   instHMIStationDriver.instsHSSPartSelect[2].lib.raw[9,5] := WSTRING#'16.18.011.321.010A';
   instHMIStationDriver.instsHSSPartSelect[2].lib.raw[9,6] := WSTRING#'16.18.008.301.030A';
   instHMIStationDriver.instsHSSPartSelect[2].lib.raw[9,7] := WSTRING#'16.18.011.321.020B';
   instHMIStationDriver.instsHSSPartSelect[2].lib.raw[10,0] := WSTRING#'';
   instHMIStationDriver.instsHSSPartSelect[2].lib.raw[10,1] := WSTRING#'C/O MATERIALS';
   instHMIStationDriver.instsHSSPartSelect[2].lib.raw[10,2] := WSTRING#'16.18.007.301.010A';
   instHMIStationDriver.instsHSSPartSelect[2].lib.raw[10,3] := WSTRING#'16.18.011.321.020B';
   instHMIStationDriver.instsHSSPartSelect[2].lib.raw[10,4] := WSTRING#'';
   instHMIStationDriver.instsHSSPartSelect[2].lib.raw[10,5] := WSTRING#'16.18.008.301.020A';
   instHMIStationDriver.instsHSSPartSelect[2].lib.raw[10,6] := WSTRING#'16.18.008.301.030A';
   instHMIStationDriver.instsHSSPartSelect[2].lib.raw[10,7] := WSTRING#'16.18.011.301.020B';
   instHMIStationDriver.instsHSSPartSelect[2].lib.raw[11,0] := WSTRING#'';
   instHMIStationDriver.instsHSSPartSelect[2].lib.raw[11,1] := WSTRING#'C/O MATERIALS';
   instHMIStationDriver.instsHSSPartSelect[2].lib.raw[11,2] := WSTRING#'16.18.008.311.010A';
   instHMIStationDriver.instsHSSPartSelect[2].lib.raw[11,3] := WSTRING#'';
   instHMIStationDriver.instsHSSPartSelect[2].lib.raw[11,4] := WSTRING#'';
   instHMIStationDriver.instsHSSPartSelect[2].lib.raw[11,5] := WSTRING#'';
   instHMIStationDriver.instsHSSPartSelect[2].lib.raw[11,6] := WSTRING#'16.18.008.301.030A';
   instHMIStationDriver.instsHSSPartSelect[2].lib.raw[11,7] := WSTRING#'16.18.008.311.020B';
   instHMIStationDriver.instsHSSPartSelect[2].lib.raw[12,0] := WSTRING#'';
   instHMIStationDriver.instsHSSPartSelect[2].lib.raw[12,1] := WSTRING#'C/O MATERIALS';
   instHMIStationDriver.instsHSSPartSelect[2].lib.raw[12,2] := WSTRING#'16.18.009.301.010A';
   instHMIStationDriver.instsHSSPartSelect[2].lib.raw[12,3] := WSTRING#'16.18.009.301.040B';
   instHMIStationDriver.instsHSSPartSelect[2].lib.raw[12,4] := WSTRING#'';
   instHMIStationDriver.instsHSSPartSelect[2].lib.raw[12,5] := WSTRING#'16.18.009.301.030A';
   instHMIStationDriver.instsHSSPartSelect[2].lib.raw[12,6] := WSTRING#'16.18.009.301.050A';
   instHMIStationDriver.instsHSSPartSelect[2].lib.raw[12,7] := WSTRING#'16.18.009.301.020B';
   instHMIStationDriver.instsHSSPartSelect[2].lib.raw[13,0] := WSTRING#'';
   instHMIStationDriver.instsHSSPartSelect[2].lib.raw[13,1] := WSTRING#'C/O MATERIALS';
   instHMIStationDriver.instsHSSPartSelect[2].lib.raw[13,2] := WSTRING#'16.18.009.311.010A';
   instHMIStationDriver.instsHSSPartSelect[2].lib.raw[13,3] := WSTRING#'';
   instHMIStationDriver.instsHSSPartSelect[2].lib.raw[13,4] := WSTRING#'';
   instHMIStationDriver.instsHSSPartSelect[2].lib.raw[13,5] := WSTRING#'16.18.009.301.030A';
   instHMIStationDriver.instsHSSPartSelect[2].lib.raw[13,6] := WSTRING#'16.18.009.301.050A';
   instHMIStationDriver.instsHSSPartSelect[2].lib.raw[13,7] := WSTRING#'16.18.009.301.040B';
   instHMIStationDriver.instsHSSPartSelect[2].lib.raw[14,0] := WSTRING#'';
   instHMIStationDriver.instsHSSPartSelect[2].lib.raw[14,1] := WSTRING#'C/O MATERIALS';
   instHMIStationDriver.instsHSSPartSelect[2].lib.raw[14,2] := WSTRING#'16.18.009.321.010A';
   instHMIStationDriver.instsHSSPartSelect[2].lib.raw[14,3] := WSTRING#'16.18.009.301.020B';
   instHMIStationDriver.instsHSSPartSelect[2].lib.raw[14,4] := WSTRING#'';
   instHMIStationDriver.instsHSSPartSelect[2].lib.raw[14,5] := WSTRING#'16.18.009.321.030A';
   instHMIStationDriver.instsHSSPartSelect[2].lib.raw[14,6] := WSTRING#'16.18.009.301.050A';
   instHMIStationDriver.instsHSSPartSelect[2].lib.raw[14,7] := WSTRING#'16.18.009.321.020B';
   instHMIStationDriver.instsHSSPartSelect[2].lib.raw[15,0] := WSTRING#'';
   instHMIStationDriver.instsHSSPartSelect[2].lib.raw[15,1] := WSTRING#'C/O MATERIALS';
   instHMIStationDriver.instsHSSPartSelect[2].lib.raw[15,2] := WSTRING#'16.18.009.321.010A';
   instHMIStationDriver.instsHSSPartSelect[2].lib.raw[15,3] := WSTRING#'16.18.009.321.020B';
   instHMIStationDriver.instsHSSPartSelect[2].lib.raw[15,4] := WSTRING#'';
   instHMIStationDriver.instsHSSPartSelect[2].lib.raw[15,5] := WSTRING#'16.18.009.321.030A';
   instHMIStationDriver.instsHSSPartSelect[2].lib.raw[15,6] := WSTRING#'16.18.009.331.050A';
   instHMIStationDriver.instsHSSPartSelect[2].lib.raw[15,7] := WSTRING#'16.18.009.301.020B';
   instHMIStationDriver.instsHSSPartSelect[2].lib.raw[16,0] := WSTRING#'';
   instHMIStationDriver.instsHSSPartSelect[2].lib.raw[16,1] := WSTRING#'C/O MATERIALS';
   instHMIStationDriver.instsHSSPartSelect[2].lib.raw[16,2] := WSTRING#'16.18.009.331.030A';
   instHMIStationDriver.instsHSSPartSelect[2].lib.raw[16,3] := WSTRING#'';
   instHMIStationDriver.instsHSSPartSelect[2].lib.raw[16,4] := WSTRING#'';
   instHMIStationDriver.instsHSSPartSelect[2].lib.raw[16,5] := WSTRING#'16.18.009.371.010A';
   instHMIStationDriver.instsHSSPartSelect[2].lib.raw[16,6] := WSTRING#'16.18.009.301.050A';
   instHMIStationDriver.instsHSSPartSelect[2].lib.raw[16,7] := WSTRING#'16.18.009.301.020B';
   instHMIStationDriver.instsHSSPartSelect[2].lib.raw[17,0] := WSTRING#'';
   instHMIStationDriver.instsHSSPartSelect[2].lib.raw[17,1] := WSTRING#'C/O MATERIALS';
   instHMIStationDriver.instsHSSPartSelect[2].lib.raw[17,2] := WSTRING#'16.18.011.301.030A';
   instHMIStationDriver.instsHSSPartSelect[2].lib.raw[17,3] := WSTRING#'16.18.011.301.040B';
   instHMIStationDriver.instsHSSPartSelect[2].lib.raw[17,4] := WSTRING#'';
   instHMIStationDriver.instsHSSPartSelect[2].lib.raw[17,5] := WSTRING#'16.18.011.301.010A';
   instHMIStationDriver.instsHSSPartSelect[2].lib.raw[17,6] := WSTRING#'16.18.008.301.030A';
   instHMIStationDriver.instsHSSPartSelect[2].lib.raw[17,7] := WSTRING#'16.18.011.301.020B';
   instHMIStationDriver.instsHSSPartSelect[2].lib.raw[18,0] := WSTRING#'';
   instHMIStationDriver.instsHSSPartSelect[2].lib.raw[18,1] := WSTRING#'C/O MATERIALS';
   instHMIStationDriver.instsHSSPartSelect[2].lib.raw[18,2] := WSTRING#'16.18.007.301.010A';
   instHMIStationDriver.instsHSSPartSelect[2].lib.raw[18,3] := WSTRING#'';
   instHMIStationDriver.instsHSSPartSelect[2].lib.raw[18,4] := WSTRING#'';
   instHMIStationDriver.instsHSSPartSelect[2].lib.raw[18,5] := WSTRING#'16.18.011.321.010A';
   instHMIStationDriver.instsHSSPartSelect[2].lib.raw[18,6] := WSTRING#'16.18.011.311.020A';
   instHMIStationDriver.instsHSSPartSelect[2].lib.raw[18,7] := WSTRING#'16.18.011.321.020B';
   instHMIStationDriver.instsHSSPartSelect[2].lib.raw[19,0] := WSTRING#'';
   instHMIStationDriver.instsHSSPartSelect[2].lib.raw[19,1] := WSTRING#'C/O MATERIALS';
   instHMIStationDriver.instsHSSPartSelect[2].lib.raw[19,2] := WSTRING#'16.18.011.321.010A';
   instHMIStationDriver.instsHSSPartSelect[2].lib.raw[19,3] := WSTRING#'16.18.011.301.020B';
   instHMIStationDriver.instsHSSPartSelect[2].lib.raw[19,4] := WSTRING#'';
   instHMIStationDriver.instsHSSPartSelect[2].lib.raw[19,5] := WSTRING#'16.18.011.301.010A';
   instHMIStationDriver.instsHSSPartSelect[2].lib.raw[19,6] := WSTRING#'16.18.011.321.030A';
   instHMIStationDriver.instsHSSPartSelect[2].lib.raw[19,7] := WSTRING#'16.18.011.321.020B';
   instHMIStationDriver.instsHSSPartSelect[2].lib.raw[20,0] := WSTRING#'';
   instHMIStationDriver.instsHSSPartSelect[2].lib.raw[20,1] := WSTRING#'C/O MATERIALS';
   instHMIStationDriver.instsHSSPartSelect[2].lib.raw[20,2] := WSTRING#'16.18.011.331.010A';
   instHMIStationDriver.instsHSSPartSelect[2].lib.raw[20,3] := WSTRING#'';
   instHMIStationDriver.instsHSSPartSelect[2].lib.raw[20,4] := WSTRING#'';
   instHMIStationDriver.instsHSSPartSelect[2].lib.raw[20,5] := WSTRING#'';
   instHMIStationDriver.instsHSSPartSelect[2].lib.raw[20,6] := WSTRING#'16.18.011.311.020A';
   instHMIStationDriver.instsHSSPartSelect[2].lib.raw[20,7] := WSTRING#'16.18.011.331.020D';
   instHMIStationDriver.instsHSSPartSelect[2].lib.raw[21,0] := WSTRING#'';
   instHMIStationDriver.instsHSSPartSelect[2].lib.raw[21,1] := WSTRING#'C/O MATERIALS';
   instHMIStationDriver.instsHSSPartSelect[2].lib.raw[21,2] := WSTRING#'16.18.012.401.010A';
   instHMIStationDriver.instsHSSPartSelect[2].lib.raw[21,3] := WSTRING#'';
   instHMIStationDriver.instsHSSPartSelect[2].lib.raw[21,4] := WSTRING#'';
   instHMIStationDriver.instsHSSPartSelect[2].lib.raw[21,5] := WSTRING#'';
   instHMIStationDriver.instsHSSPartSelect[2].lib.raw[21,6] := WSTRING#'16.18.014.411.030A';
   instHMIStationDriver.instsHSSPartSelect[2].lib.raw[21,7] := WSTRING#'16.18.012.401.020A';
   instHMIStationDriver.instsHSSPartSelect[2].lib.raw[22,0] := WSTRING#'';
   instHMIStationDriver.instsHSSPartSelect[2].lib.raw[22,1] := WSTRING#'C/O MATERIALS';
   instHMIStationDriver.instsHSSPartSelect[2].lib.raw[22,2] := WSTRING#'16.18.012.411.010A';
   instHMIStationDriver.instsHSSPartSelect[2].lib.raw[22,3] := WSTRING#'';
   instHMIStationDriver.instsHSSPartSelect[2].lib.raw[22,4] := WSTRING#'';
   instHMIStationDriver.instsHSSPartSelect[2].lib.raw[22,5] := WSTRING#'';
   instHMIStationDriver.instsHSSPartSelect[2].lib.raw[22,6] := WSTRING#'16.18.014.411.030A';
   instHMIStationDriver.instsHSSPartSelect[2].lib.raw[22,7] := WSTRING#'16.18.012.411.020B';
   instHMIStationDriver.instsHSSPartSelect[2].lib.raw[23,0] := WSTRING#'';
   instHMIStationDriver.instsHSSPartSelect[2].lib.raw[23,1] := WSTRING#'C/O MATERIALS';
   instHMIStationDriver.instsHSSPartSelect[2].lib.raw[23,2] := WSTRING#'16.18.014.411.010A';
   instHMIStationDriver.instsHSSPartSelect[2].lib.raw[23,3] := WSTRING#'';
   instHMIStationDriver.instsHSSPartSelect[2].lib.raw[23,4] := WSTRING#'';
   instHMIStationDriver.instsHSSPartSelect[2].lib.raw[23,5] := WSTRING#'';
   instHMIStationDriver.instsHSSPartSelect[2].lib.raw[23,6] := WSTRING#'16.18.014.411.030A';
   instHMIStationDriver.instsHSSPartSelect[2].lib.raw[23,7] := WSTRING#'16.18.012.401.020A';
   instHMIStationDriver.instsHSSPartSelect[2].lib.raw[24,0] := WSTRING#'';
   instHMIStationDriver.instsHSSPartSelect[2].lib.raw[24,1] := WSTRING#'C/O MATERIALS';
   instHMIStationDriver.instsHSSPartSelect[2].lib.raw[24,2] := WSTRING#'16.18.012.431.010A';
   instHMIStationDriver.instsHSSPartSelect[2].lib.raw[24,3] := WSTRING#'';
   instHMIStationDriver.instsHSSPartSelect[2].lib.raw[24,4] := WSTRING#'';
   instHMIStationDriver.instsHSSPartSelect[2].lib.raw[24,5] := WSTRING#'';
   instHMIStationDriver.instsHSSPartSelect[2].lib.raw[24,6] := WSTRING#'16.18.014.411.030A';
   instHMIStationDriver.instsHSSPartSelect[2].lib.raw[24,7] := WSTRING#'16.18.012.411.020B';
   instHMIStationDriver.instsHSSPartSelect[2].lib.raw[25,0] := WSTRING#'';
   instHMIStationDriver.instsHSSPartSelect[2].lib.raw[25,1] := WSTRING#'C/O MATERIALS';
   instHMIStationDriver.instsHSSPartSelect[2].lib.raw[25,2] := WSTRING#'16.18.012.441.010A';
   instHMIStationDriver.instsHSSPartSelect[2].lib.raw[25,3] := WSTRING#'';
   instHMIStationDriver.instsHSSPartSelect[2].lib.raw[25,4] := WSTRING#'';
   instHMIStationDriver.instsHSSPartSelect[2].lib.raw[25,5] := WSTRING#'';
   instHMIStationDriver.instsHSSPartSelect[2].lib.raw[25,6] := WSTRING#'16.18.013.411.030A';
   instHMIStationDriver.instsHSSPartSelect[2].lib.raw[25,7] := WSTRING#'16.18.011.321.020B';
   instHMIStationDriver.instsHSSPartSelect[2].lib.raw[26,0] := WSTRING#'';
   instHMIStationDriver.instsHSSPartSelect[2].lib.raw[26,1] := WSTRING#'C/O MATERIALS';
   instHMIStationDriver.instsHSSPartSelect[2].lib.raw[26,2] := WSTRING#'16.18.013.411.010A';
   instHMIStationDriver.instsHSSPartSelect[2].lib.raw[26,3] := WSTRING#'';
   instHMIStationDriver.instsHSSPartSelect[2].lib.raw[26,4] := WSTRING#'';
   instHMIStationDriver.instsHSSPartSelect[2].lib.raw[26,5] := WSTRING#'';
   instHMIStationDriver.instsHSSPartSelect[2].lib.raw[26,6] := WSTRING#'16.18.013.411.030A';
   instHMIStationDriver.instsHSSPartSelect[2].lib.raw[26,7] := WSTRING#'16.18.013.411.020B';
   instHMIStationDriver.instsHSSPartSelect[2].lib.raw[27,0] := WSTRING#'';
   instHMIStationDriver.instsHSSPartSelect[2].lib.raw[27,1] := WSTRING#'C/O MATERIALS';
   instHMIStationDriver.instsHSSPartSelect[2].lib.raw[27,2] := WSTRING#'16.18.013.421.010A';
   instHMIStationDriver.instsHSSPartSelect[2].lib.raw[27,3] := WSTRING#'';
   instHMIStationDriver.instsHSSPartSelect[2].lib.raw[27,4] := WSTRING#'';
   instHMIStationDriver.instsHSSPartSelect[2].lib.raw[27,5] := WSTRING#'';
   instHMIStationDriver.instsHSSPartSelect[2].lib.raw[27,6] := WSTRING#'16.18.013.411.030A';
   instHMIStationDriver.instsHSSPartSelect[2].lib.raw[27,7] := WSTRING#'16.18.011.301.040B';
   instHMIStationDriver.instsHSSPartSelect[2].lib.raw[28,0] := WSTRING#'';
   instHMIStationDriver.instsHSSPartSelect[2].lib.raw[28,1] := WSTRING#'C/O MATERIALS';
   instHMIStationDriver.instsHSSPartSelect[2].lib.raw[28,2] := WSTRING#'16.18.015.421.010A';
   instHMIStationDriver.instsHSSPartSelect[2].lib.raw[28,3] := WSTRING#'';
   instHMIStationDriver.instsHSSPartSelect[2].lib.raw[28,4] := WSTRING#'';
   instHMIStationDriver.instsHSSPartSelect[2].lib.raw[28,5] := WSTRING#'';
   instHMIStationDriver.instsHSSPartSelect[2].lib.raw[28,6] := WSTRING#'16.18.015.401.010A';
   instHMIStationDriver.instsHSSPartSelect[2].lib.raw[28,7] := WSTRING#'16.18.015.421.020B';
   instHMIStationDriver.instsHSSPartSelect[2].lib.raw[29,0] := WSTRING#'';
   instHMIStationDriver.instsHSSPartSelect[2].lib.raw[29,1] := WSTRING#'C/O MATERIALS';
   instHMIStationDriver.instsHSSPartSelect[2].lib.raw[29,2] := WSTRING#'16.18.015.411.010A';
   instHMIStationDriver.instsHSSPartSelect[2].lib.raw[29,3] := WSTRING#'';
   instHMIStationDriver.instsHSSPartSelect[2].lib.raw[29,4] := WSTRING#'';
   instHMIStationDriver.instsHSSPartSelect[2].lib.raw[29,5] := WSTRING#'';
   instHMIStationDriver.instsHSSPartSelect[2].lib.raw[29,6] := WSTRING#'16.18.015.411.030A';
   instHMIStationDriver.instsHSSPartSelect[2].lib.raw[29,7] := WSTRING#'16.18.015.411.020B';
   instHMIStationDriver.instsHSSPartSelect[2].lib.raw[30,0] := WSTRING#'';
   instHMIStationDriver.instsHSSPartSelect[2].lib.raw[30,1] := WSTRING#'C/O MATERIALS';
   instHMIStationDriver.instsHSSPartSelect[2].lib.raw[30,2] := WSTRING#'16.18.018.401.010A';
   instHMIStationDriver.instsHSSPartSelect[2].lib.raw[30,3] := WSTRING#'';
   instHMIStationDriver.instsHSSPartSelect[2].lib.raw[30,4] := WSTRING#'';
   instHMIStationDriver.instsHSSPartSelect[2].lib.raw[30,5] := WSTRING#'';
   instHMIStationDriver.instsHSSPartSelect[2].lib.raw[30,6] := WSTRING#'16.18.015.401.010A';
   instHMIStationDriver.instsHSSPartSelect[2].lib.raw[30,7] := WSTRING#'16.18.018.401.020B';
   instHMIStationDriver.instsHSSPartSelect[2].lib.raw[31,0] := WSTRING#'';
   instHMIStationDriver.instsHSSPartSelect[2].lib.raw[31,1] := WSTRING#'C/O MATERIALS';
   instHMIStationDriver.instsHSSPartSelect[2].lib.raw[31,2] := WSTRING#'16.18.018.421.010B';
   instHMIStationDriver.instsHSSPartSelect[2].lib.raw[31,3] := WSTRING#'';
   instHMIStationDriver.instsHSSPartSelect[2].lib.raw[31,4] := WSTRING#'';
   instHMIStationDriver.instsHSSPartSelect[2].lib.raw[31,5] := WSTRING#'';
   instHMIStationDriver.instsHSSPartSelect[2].lib.raw[31,6] := WSTRING#'16.18.015.411.030A';
   instHMIStationDriver.instsHSSPartSelect[2].lib.raw[31,7] := WSTRING#'16.18.015.411.020B';
   instHMIStationDriver.instsHSSPartSelect[2].lib.raw[32,0] := WSTRING#'';
   instHMIStationDriver.instsHSSPartSelect[2].lib.raw[32,1] := WSTRING#'C/O MATERIALS';
   instHMIStationDriver.instsHSSPartSelect[2].lib.raw[32,2] := WSTRING#'16.18.018.401.010A';
   instHMIStationDriver.instsHSSPartSelect[2].lib.raw[32,3] := WSTRING#'';
   instHMIStationDriver.instsHSSPartSelect[2].lib.raw[32,4] := WSTRING#'';
   instHMIStationDriver.instsHSSPartSelect[2].lib.raw[32,5] := WSTRING#'';
   instHMIStationDriver.instsHSSPartSelect[2].lib.raw[32,6] := WSTRING#'16.18.015.411.030A';
   instHMIStationDriver.instsHSSPartSelect[2].lib.raw[32,7] := WSTRING#'16.18.018.401.020B';
   instHMIStationDriver.instsHSSPartSelect[2].lib.raw[33,0] := WSTRING#'';
   instHMIStationDriver.instsHSSPartSelect[2].lib.raw[33,1] := WSTRING#'C/O MATERIALS';
   instHMIStationDriver.instsHSSPartSelect[2].lib.raw[33,2] := WSTRING#'16.18.017.301.030A';
   instHMIStationDriver.instsHSSPartSelect[2].lib.raw[33,3] := WSTRING#'16.18.017.301.020A';
   instHMIStationDriver.instsHSSPartSelect[2].lib.raw[33,4] := WSTRING#'';
   instHMIStationDriver.instsHSSPartSelect[2].lib.raw[33,5] := WSTRING#'16.18.017.301.010A';
   instHMIStationDriver.instsHSSPartSelect[2].lib.raw[33,6] := WSTRING#'16.18.017.301.050A';
   instHMIStationDriver.instsHSSPartSelect[2].lib.raw[33,7] := WSTRING#'16.18.017.301.040A';
   instHMIStationDriver.instsHSSPartSelect[2].lib.raw[34,0] := WSTRING#'';
   instHMIStationDriver.instsHSSPartSelect[2].lib.raw[34,1] := WSTRING#'C/O MATERIALS';
   instHMIStationDriver.instsHSSPartSelect[2].lib.raw[34,2] := WSTRING#'16.18.017.301.030A';
   instHMIStationDriver.instsHSSPartSelect[2].lib.raw[34,3] := WSTRING#'';
   instHMIStationDriver.instsHSSPartSelect[2].lib.raw[34,4] := WSTRING#'';
   instHMIStationDriver.instsHSSPartSelect[2].lib.raw[34,5] := WSTRING#'16.18.017.311.010A';
   instHMIStationDriver.instsHSSPartSelect[2].lib.raw[34,6] := WSTRING#'16.18.017.301.050A';
   instHMIStationDriver.instsHSSPartSelect[2].lib.raw[34,7] := WSTRING#'16.18.017.301.040A';
   instHMIStationDriver.instsHSSPartSelect[2].lib.raw[35,0] := WSTRING#'';
   instHMIStationDriver.instsHSSPartSelect[2].lib.raw[35,1] := WSTRING#'C/O MATERIALS';
   instHMIStationDriver.instsHSSPartSelect[2].lib.raw[35,2] := WSTRING#'16.18.017.321.010A';
   instHMIStationDriver.instsHSSPartSelect[2].lib.raw[35,3] := WSTRING#'';
   instHMIStationDriver.instsHSSPartSelect[2].lib.raw[35,4] := WSTRING#'';
   instHMIStationDriver.instsHSSPartSelect[2].lib.raw[35,5] := WSTRING#'';
   instHMIStationDriver.instsHSSPartSelect[2].lib.raw[35,6] := WSTRING#'16.18.017.301.050A';
   instHMIStationDriver.instsHSSPartSelect[2].lib.raw[35,7] := WSTRING#'16.18.017.321.020A';
   instHMIStationDriver.instsHSSPartSelect[2].lib.raw[36,0] := WSTRING#'';
   instHMIStationDriver.instsHSSPartSelect[2].lib.raw[36,1] := WSTRING#'C/O MATERIALS';
   instHMIStationDriver.instsHSSPartSelect[2].lib.raw[36,2] := WSTRING#'16.18.018.401.010A';
   instHMIStationDriver.instsHSSPartSelect[2].lib.raw[36,3] := WSTRING#'';
   instHMIStationDriver.instsHSSPartSelect[2].lib.raw[36,4] := WSTRING#'';
   instHMIStationDriver.instsHSSPartSelect[2].lib.raw[36,5] := WSTRING#'';
   instHMIStationDriver.instsHSSPartSelect[2].lib.raw[36,6] := WSTRING#'16.18.018.401.030A';
   instHMIStationDriver.instsHSSPartSelect[2].lib.raw[36,7] := WSTRING#'16.18.018.401.020B';
   instHMIStationDriver.instsHSSPartSelect[2].lib.raw[37,0] := WSTRING#'';
   instHMIStationDriver.instsHSSPartSelect[2].lib.raw[37,1] := WSTRING#'C/O MATERIALS';
   instHMIStationDriver.instsHSSPartSelect[2].lib.raw[37,2] := WSTRING#'16.18.015.411.010A';
   instHMIStationDriver.instsHSSPartSelect[2].lib.raw[37,3] := WSTRING#'';
   instHMIStationDriver.instsHSSPartSelect[2].lib.raw[37,4] := WSTRING#'';
   instHMIStationDriver.instsHSSPartSelect[2].lib.raw[37,5] := WSTRING#'';
   instHMIStationDriver.instsHSSPartSelect[2].lib.raw[37,6] := WSTRING#'16.18.018.401.030A';
   instHMIStationDriver.instsHSSPartSelect[2].lib.raw[37,7] := WSTRING#'16.18.015.411.020B';
   instHMIStationDriver.instsHSSPartSelect[2].lib.raw[38,0] := WSTRING#'';
   instHMIStationDriver.instsHSSPartSelect[2].lib.raw[38,1] := WSTRING#'C/O MATERIALS';
   instHMIStationDriver.instsHSSPartSelect[2].lib.raw[38,2] := WSTRING#'16.18.018.411.010A';
   instHMIStationDriver.instsHSSPartSelect[2].lib.raw[38,3] := WSTRING#'';
   instHMIStationDriver.instsHSSPartSelect[2].lib.raw[38,4] := WSTRING#'';
   instHMIStationDriver.instsHSSPartSelect[2].lib.raw[38,5] := WSTRING#'';
   instHMIStationDriver.instsHSSPartSelect[2].lib.raw[38,6] := WSTRING#'16.18.018.401.030A';
   instHMIStationDriver.instsHSSPartSelect[2].lib.raw[38,7] := WSTRING#'16.18.018.401.020B';
   instHMIStationDriver.instsHSSPartSelect[2].lib.raw[39,0] := WSTRING#'';
   instHMIStationDriver.instsHSSPartSelect[2].lib.raw[39,1] := WSTRING#'C/O MATERIALS';
   instHMIStationDriver.instsHSSPartSelect[2].lib.raw[39,2] := WSTRING#'16.18.018.421.010B';
   instHMIStationDriver.instsHSSPartSelect[2].lib.raw[39,3] := WSTRING#'';
   instHMIStationDriver.instsHSSPartSelect[2].lib.raw[39,4] := WSTRING#'';
   instHMIStationDriver.instsHSSPartSelect[2].lib.raw[39,5] := WSTRING#'';
   instHMIStationDriver.instsHSSPartSelect[2].lib.raw[39,6] := WSTRING#'16.18.018.401.030A';
   instHMIStationDriver.instsHSSPartSelect[2].lib.raw[39,7] := WSTRING#'16.18.015.411.020B';
   instHMIStationDriver.instsHSSPartSelect[2].lib.raw[40,0] := WSTRING#'';
   instHMIStationDriver.instsHSSPartSelect[2].lib.raw[40,1] := WSTRING#'C/O MATERIALS';
   instHMIStationDriver.instsHSSPartSelect[2].lib.raw[40,2] := WSTRING#'16.18.008.301.010A';
   instHMIStationDriver.instsHSSPartSelect[2].lib.raw[40,3] := WSTRING#'16.18.011.321.020B';
   instHMIStationDriver.instsHSSPartSelect[2].lib.raw[40,4] := WSTRING#'';
   instHMIStationDriver.instsHSSPartSelect[2].lib.raw[40,5] := WSTRING#'16.18.011.321.010A';
   instHMIStationDriver.instsHSSPartSelect[2].lib.raw[40,6] := WSTRING#'16.18.011.311.020A';
   instHMIStationDriver.instsHSSPartSelect[2].lib.raw[40,7] := WSTRING#'16.18.012.401.020A';
   instHMIStationDriver.instsHSSPartSelect[2].lib.raw[41,0] := WSTRING#'';
   instHMIStationDriver.instsHSSPartSelect[2].lib.raw[41,1] := WSTRING#'C/O MATERIALS';
   instHMIStationDriver.instsHSSPartSelect[2].lib.raw[41,2] := WSTRING#'16.32.606.311.040B';
   instHMIStationDriver.instsHSSPartSelect[2].lib.raw[41,3] := WSTRING#'16.32.606.311.070A';
   instHMIStationDriver.instsHSSPartSelect[2].lib.raw[41,4] := WSTRING#'';
   instHMIStationDriver.instsHSSPartSelect[2].lib.raw[41,5] := WSTRING#'16.32.606.311.050B';
   instHMIStationDriver.instsHSSPartSelect[2].lib.raw[41,6] := WSTRING#'16.32.606.311.010F';
   instHMIStationDriver.instsHSSPartSelect[2].lib.raw[41,7] := WSTRING#'16.32.606.311.060A';
   instHMIStationDriver.instsHSSPartSelect[2].lib.raw[42,0] := WSTRING#'';
   instHMIStationDriver.instsHSSPartSelect[2].lib.raw[42,1] := WSTRING#'C/O MATERIALS';
   instHMIStationDriver.instsHSSPartSelect[2].lib.raw[42,2] := WSTRING#'16.32.112.054.041A';
   instHMIStationDriver.instsHSSPartSelect[2].lib.raw[42,3] := WSTRING#'';
   instHMIStationDriver.instsHSSPartSelect[2].lib.raw[42,4] := WSTRING#'';
   instHMIStationDriver.instsHSSPartSelect[2].lib.raw[42,5] := WSTRING#'16.32.112.057.010A';
   instHMIStationDriver.instsHSSPartSelect[2].lib.raw[42,6] := WSTRING#'16.32.112.553.100D';
   instHMIStationDriver.instsHSSPartSelect[2].lib.raw[42,7] := WSTRING#'16.32.806.315.001A';
   instHMIStationDriver.instsHSSPartSelect[2].lib.raw[43,0] := WSTRING#'';
   instHMIStationDriver.instsHSSPartSelect[2].lib.raw[43,1] := WSTRING#'C/O MATERIALS';
   instHMIStationDriver.instsHSSPartSelect[2].lib.raw[43,2] := WSTRING#'16.08.211.806.020A';
   instHMIStationDriver.instsHSSPartSelect[2].lib.raw[43,3] := WSTRING#'';
   instHMIStationDriver.instsHSSPartSelect[2].lib.raw[43,4] := WSTRING#'';
   instHMIStationDriver.instsHSSPartSelect[2].lib.raw[43,5] := WSTRING#'';
   instHMIStationDriver.instsHSSPartSelect[2].lib.raw[43,6] := WSTRING#'16.08.208.631.000F';
   instHMIStationDriver.instsHSSPartSelect[2].lib.raw[43,7] := WSTRING#'16.08.216.315.000A';
   instHMIStationDriver.instsHSSPartSelect[2].lib.raw[44,0] := WSTRING#'';
   instHMIStationDriver.instsHSSPartSelect[2].lib.raw[44,1] := WSTRING#'C/O MATERIALS';
   instHMIStationDriver.instsHSSPartSelect[2].lib.raw[44,2] := WSTRING#'16.08.208.041.000A';
   instHMIStationDriver.instsHSSPartSelect[2].lib.raw[44,3] := WSTRING#'16.08.208.031.020C';
   instHMIStationDriver.instsHSSPartSelect[2].lib.raw[44,4] := WSTRING#'';
   instHMIStationDriver.instsHSSPartSelect[2].lib.raw[44,5] := WSTRING#'16.08.211.291.000A';
   instHMIStationDriver.instsHSSPartSelect[2].lib.raw[44,6] := WSTRING#'16.08.208.661.000F';
   instHMIStationDriver.instsHSSPartSelect[2].lib.raw[44,7] := WSTRING#'16.08.208.651.010B';
   instHMIStationDriver.instsHSSPartSelect[2].lib.raw[45,0] := WSTRING#'';
   instHMIStationDriver.instsHSSPartSelect[2].lib.raw[45,1] := WSTRING#'C/O MATERIALS';
   instHMIStationDriver.instsHSSPartSelect[2].lib.raw[45,2] := WSTRING#'';
   instHMIStationDriver.instsHSSPartSelect[2].lib.raw[45,3] := WSTRING#'';
   instHMIStationDriver.instsHSSPartSelect[2].lib.raw[45,4] := WSTRING#'';
   instHMIStationDriver.instsHSSPartSelect[2].lib.raw[45,5] := WSTRING#'';
   instHMIStationDriver.instsHSSPartSelect[2].lib.raw[45,6] := WSTRING#'';
   instHMIStationDriver.instsHSSPartSelect[2].lib.raw[45,7] := WSTRING#'';
   instHMIStationDriver.instsHSSPartSelect[2].lib.raw[46,0] := WSTRING#'';
   instHMIStationDriver.instsHSSPartSelect[2].lib.raw[46,1] := WSTRING#'C/O MATERIALS';
   instHMIStationDriver.instsHSSPartSelect[2].lib.raw[46,2] := WSTRING#'';
   instHMIStationDriver.instsHSSPartSelect[2].lib.raw[46,3] := WSTRING#'';
   instHMIStationDriver.instsHSSPartSelect[2].lib.raw[46,4] := WSTRING#'';
   instHMIStationDriver.instsHSSPartSelect[2].lib.raw[46,5] := WSTRING#'';
   instHMIStationDriver.instsHSSPartSelect[2].lib.raw[46,6] := WSTRING#'';
   instHMIStationDriver.instsHSSPartSelect[2].lib.raw[46,7] := WSTRING#'';
   instHMIStationDriver.instsHSSPartSelect[2].lib.raw[47,0] := WSTRING#'';
   instHMIStationDriver.instsHSSPartSelect[2].lib.raw[47,1] := WSTRING#'C/O MATERIALS';
   instHMIStationDriver.instsHSSPartSelect[2].lib.raw[47,2] := WSTRING#'';
   instHMIStationDriver.instsHSSPartSelect[2].lib.raw[47,3] := WSTRING#'';
   instHMIStationDriver.instsHSSPartSelect[2].lib.raw[47,4] := WSTRING#'';
   instHMIStationDriver.instsHSSPartSelect[2].lib.raw[47,5] := WSTRING#'';
   instHMIStationDriver.instsHSSPartSelect[2].lib.raw[47,6] := WSTRING#'';
   instHMIStationDriver.instsHSSPartSelect[2].lib.raw[47,7] := WSTRING#'';
   instHMIStationDriver.instsHSSPartSelect[2].lib.raw[48,0] := WSTRING#'';
   instHMIStationDriver.instsHSSPartSelect[2].lib.raw[48,1] := WSTRING#'C/O MATERIALS';
   instHMIStationDriver.instsHSSPartSelect[2].lib.raw[48,2] := WSTRING#'';
   instHMIStationDriver.instsHSSPartSelect[2].lib.raw[48,3] := WSTRING#'';
   instHMIStationDriver.instsHSSPartSelect[2].lib.raw[48,4] := WSTRING#'';
   instHMIStationDriver.instsHSSPartSelect[2].lib.raw[48,5] := WSTRING#'';
   instHMIStationDriver.instsHSSPartSelect[2].lib.raw[48,6] := WSTRING#'';
   instHMIStationDriver.instsHSSPartSelect[2].lib.raw[48,7] := WSTRING#'';
   instHMIStationDriver.instsHSSPartSelect[2].lib.raw[49,0] := WSTRING#'';
   instHMIStationDriver.instsHSSPartSelect[2].lib.raw[49,1] := WSTRING#'C/O MATERIALS';
   instHMIStationDriver.instsHSSPartSelect[2].lib.raw[49,2] := WSTRING#'';
   instHMIStationDriver.instsHSSPartSelect[2].lib.raw[49,3] := WSTRING#'';
   instHMIStationDriver.instsHSSPartSelect[2].lib.raw[49,4] := WSTRING#'';
   instHMIStationDriver.instsHSSPartSelect[2].lib.raw[49,5] := WSTRING#'';
   instHMIStationDriver.instsHSSPartSelect[2].lib.raw[49,6] := WSTRING#'';
   instHMIStationDriver.instsHSSPartSelect[2].lib.raw[49,7] := WSTRING#'';
   instHMIStationDriver.instsHSSPartSelect[3].recipeNum := 6;
   instHMIStationDriver.instsHSSPartSelect[3].lib.size := 11;
   instHMIStationDriver.instsHSSPartSelect[3].lib.wip[0] := WSTRING#'16.08.211.801.700B$LDPF Stuffed Shell 1 box longs only';
   instHMIStationDriver.instsHSSPartSelect[3].lib.wip[1] := WSTRING#'16.32.307.322.210A$LVolvo - ASSY INLET - SUB 8 Unformed';
   instHMIStationDriver.instsHSSPartSelect[3].lib.wip[2] := WSTRING#'16.32.112.311.001A$LSA SCR CANNING UNFORMED';
   instHMIStationDriver.instsHSSPartSelect[3].lib.wip[3] := WSTRING#'16.32.112.553.300C$LSA SCR CANNING A700 UNFORMED';
   instHMIStationDriver.instsHSSPartSelect[3].lib.wip[4] := WSTRING#'16.32.112.304.008A$LASSY SCR CANNING FORMED';
   instHMIStationDriver.instsHSSPartSelect[3].lib.wip[5] := WSTRING#'16.32.112.516.000G$LASSY DPF CANNING A700';
   instHMIStationDriver.instsHSSPartSelect[3].lib.wip[6] := WSTRING#'16.32.112.543.000E$LASSY DOC CANNING A700';
   instHMIStationDriver.instsHSSPartSelect[3].lib.wip[7] := WSTRING#'16.08.216.751.100A$LSA Sleeved SCR 2016';
   instHMIStationDriver.instsHSSPartSelect[3].lib.wip[8] := WSTRING#'16.08.208.651.000G$LStuffed Shell SCR- NGK';
   instHMIStationDriver.instsHSSPartSelect[3].lib.wip[9] := WSTRING#'16.08.211.806.400B$LSA DPF Stuffed Shell';
   instHMIStationDriver.instsHSSPartSelect[3].lib.wip[10] := WSTRING#'16.08.216.806.400A$L DPF Sleeved 2016';
   instHMIStationDriver.instsHSSPartSelect[3].lib.wip[11] := WSTRING#'';
   instHMIStationDriver.instsHSSPartSelect[3].lib.wip[12] := WSTRING#'';
   instHMIStationDriver.instsHSSPartSelect[3].lib.wip[13] := WSTRING#'';
   instHMIStationDriver.instsHSSPartSelect[3].lib.wip[14] := WSTRING#'';
   instHMIStationDriver.instsHSSPartSelect[3].lib.wip[15] := WSTRING#'';
   instHMIStationDriver.instsHSSPartSelect[3].lib.wip[16] := WSTRING#'';
   instHMIStationDriver.instsHSSPartSelect[3].lib.wip[17] := WSTRING#'';
   instHMIStationDriver.instsHSSPartSelect[3].lib.wip[18] := WSTRING#'';
   instHMIStationDriver.instsHSSPartSelect[3].lib.wip[19] := WSTRING#'';
   instHMIStationDriver.instsHSSPartSelect[3].lib.wip[20] := WSTRING#'';
   instHMIStationDriver.instsHSSPartSelect[3].lib.wip[21] := WSTRING#'';
   instHMIStationDriver.instsHSSPartSelect[3].lib.wip[22] := WSTRING#'';
   instHMIStationDriver.instsHSSPartSelect[3].lib.wip[23] := WSTRING#'';
   instHMIStationDriver.instsHSSPartSelect[3].lib.wip[24] := WSTRING#'';
   instHMIStationDriver.instsHSSPartSelect[3].lib.wip[25] := WSTRING#'';
   instHMIStationDriver.instsHSSPartSelect[3].lib.wip[26] := WSTRING#'';
   instHMIStationDriver.instsHSSPartSelect[3].lib.wip[27] := WSTRING#'';
   instHMIStationDriver.instsHSSPartSelect[3].lib.wip[28] := WSTRING#'';
   instHMIStationDriver.instsHSSPartSelect[3].lib.wip[29] := WSTRING#'';
   instHMIStationDriver.instsHSSPartSelect[3].lib.wip[30] := WSTRING#'';
   instHMIStationDriver.instsHSSPartSelect[3].lib.wip[31] := WSTRING#'';
   instHMIStationDriver.instsHSSPartSelect[3].lib.wip[32] := WSTRING#'';
   instHMIStationDriver.instsHSSPartSelect[3].lib.wip[33] := WSTRING#'';
   instHMIStationDriver.instsHSSPartSelect[3].lib.wip[34] := WSTRING#'';
   instHMIStationDriver.instsHSSPartSelect[3].lib.wip[35] := WSTRING#'';
   instHMIStationDriver.instsHSSPartSelect[3].lib.wip[36] := WSTRING#'';
   instHMIStationDriver.instsHSSPartSelect[3].lib.wip[37] := WSTRING#'';
   instHMIStationDriver.instsHSSPartSelect[3].lib.wip[38] := WSTRING#'';
   instHMIStationDriver.instsHSSPartSelect[3].lib.wip[39] := WSTRING#'';
   instHMIStationDriver.instsHSSPartSelect[3].lib.wip[40] := WSTRING#'';
   instHMIStationDriver.instsHSSPartSelect[3].lib.wip[41] := WSTRING#'';
   instHMIStationDriver.instsHSSPartSelect[3].lib.wip[42] := WSTRING#'';
   instHMIStationDriver.instsHSSPartSelect[3].lib.wip[43] := WSTRING#'';
   instHMIStationDriver.instsHSSPartSelect[3].lib.wip[44] := WSTRING#'';
   instHMIStationDriver.instsHSSPartSelect[3].lib.wip[45] := WSTRING#'';
   instHMIStationDriver.instsHSSPartSelect[3].lib.wip[46] := WSTRING#'';
   instHMIStationDriver.instsHSSPartSelect[3].lib.wip[47] := WSTRING#'';
   instHMIStationDriver.instsHSSPartSelect[3].lib.wip[48] := WSTRING#'';
   instHMIStationDriver.instsHSSPartSelect[3].lib.wip[49] := WSTRING#'';
   instHMIStationDriver.instsHSSPartSelect[3].lib.raw[0,0] := WSTRING#'';
   instHMIStationDriver.instsHSSPartSelect[3].lib.raw[0,1] := WSTRING#'C/O MATERIALS';
   instHMIStationDriver.instsHSSPartSelect[3].lib.raw[0,2] := WSTRING#'16.08.211.801.020A';
   instHMIStationDriver.instsHSSPartSelect[3].lib.raw[0,3] := WSTRING#'';
   instHMIStationDriver.instsHSSPartSelect[3].lib.raw[0,4] := WSTRING#'';
   instHMIStationDriver.instsHSSPartSelect[3].lib.raw[0,5] := WSTRING#'';
   instHMIStationDriver.instsHSSPartSelect[3].lib.raw[0,6] := WSTRING#'16.08.208.631.000F';
   instHMIStationDriver.instsHSSPartSelect[3].lib.raw[0,7] := WSTRING#'16.08.216.315.002A';
   instHMIStationDriver.instsHSSPartSelect[3].lib.raw[1,0] := WSTRING#'';
   instHMIStationDriver.instsHSSPartSelect[3].lib.raw[1,1] := WSTRING#'C/O MATERIALS';
   instHMIStationDriver.instsHSSPartSelect[3].lib.raw[1,2] := WSTRING#'16.32.307.211.150B';
   instHMIStationDriver.instsHSSPartSelect[3].lib.raw[1,3] := WSTRING#'';
   instHMIStationDriver.instsHSSPartSelect[3].lib.raw[1,4] := WSTRING#'';
   instHMIStationDriver.instsHSSPartSelect[3].lib.raw[1,5] := WSTRING#'';
   instHMIStationDriver.instsHSSPartSelect[3].lib.raw[1,6] := WSTRING#'16.32.307.211.170B';
   instHMIStationDriver.instsHSSPartSelect[3].lib.raw[1,7] := WSTRING#'16.32.307.461.160A';
   instHMIStationDriver.instsHSSPartSelect[3].lib.raw[2,0] := WSTRING#'';
   instHMIStationDriver.instsHSSPartSelect[3].lib.raw[2,1] := WSTRING#'C/O MATERIALS';
   instHMIStationDriver.instsHSSPartSelect[3].lib.raw[2,2] := WSTRING#'16.32.112.054.041A';
   instHMIStationDriver.instsHSSPartSelect[3].lib.raw[2,3] := WSTRING#'';
   instHMIStationDriver.instsHSSPartSelect[3].lib.raw[2,4] := WSTRING#'';
   instHMIStationDriver.instsHSSPartSelect[3].lib.raw[2,5] := WSTRING#'16.32.112.057.010A';
   instHMIStationDriver.instsHSSPartSelect[3].lib.raw[2,6] := WSTRING#'16.32.112.553.100D';
   instHMIStationDriver.instsHSSPartSelect[3].lib.raw[2,7] := WSTRING#'16.32.806.315.001A';
   instHMIStationDriver.instsHSSPartSelect[3].lib.raw[3,0] := WSTRING#'';
   instHMIStationDriver.instsHSSPartSelect[3].lib.raw[3,1] := WSTRING#'C/O MATERIALS';
   instHMIStationDriver.instsHSSPartSelect[3].lib.raw[3,2] := WSTRING#'16.32.112.553.010A';
   instHMIStationDriver.instsHSSPartSelect[3].lib.raw[3,3] := WSTRING#'';
   instHMIStationDriver.instsHSSPartSelect[3].lib.raw[3,4] := WSTRING#'';
   instHMIStationDriver.instsHSSPartSelect[3].lib.raw[3,5] := WSTRING#'16.32.112.553.020A';
   instHMIStationDriver.instsHSSPartSelect[3].lib.raw[3,6] := WSTRING#'16.32.112.553.100D';
   instHMIStationDriver.instsHSSPartSelect[3].lib.raw[3,7] := WSTRING#'16.32.806.315.001A';
   instHMIStationDriver.instsHSSPartSelect[3].lib.raw[4,0] := WSTRING#'';
   instHMIStationDriver.instsHSSPartSelect[3].lib.raw[4,1] := WSTRING#'C/O MATERIALS';
   instHMIStationDriver.instsHSSPartSelect[3].lib.raw[4,2] := WSTRING#'16.32.112.054.041A';
   instHMIStationDriver.instsHSSPartSelect[3].lib.raw[4,3] := WSTRING#'';
   instHMIStationDriver.instsHSSPartSelect[3].lib.raw[4,4] := WSTRING#'';
   instHMIStationDriver.instsHSSPartSelect[3].lib.raw[4,5] := WSTRING#'16.32.112.057.010A';
   instHMIStationDriver.instsHSSPartSelect[3].lib.raw[4,6] := WSTRING#'16.32.112.553.100D';
   instHMIStationDriver.instsHSSPartSelect[3].lib.raw[4,7] := WSTRING#'16.32.806.315.001A';
   instHMIStationDriver.instsHSSPartSelect[3].lib.raw[5,0] := WSTRING#'';
   instHMIStationDriver.instsHSSPartSelect[3].lib.raw[5,1] := WSTRING#'C/O MATERIALS';
   instHMIStationDriver.instsHSSPartSelect[3].lib.raw[5,2] := WSTRING#'16.32.112.536.010A';
   instHMIStationDriver.instsHSSPartSelect[3].lib.raw[5,3] := WSTRING#'';
   instHMIStationDriver.instsHSSPartSelect[3].lib.raw[5,4] := WSTRING#'';
   instHMIStationDriver.instsHSSPartSelect[3].lib.raw[5,5] := WSTRING#'';
   instHMIStationDriver.instsHSSPartSelect[3].lib.raw[5,6] := WSTRING#'16.32.112.516.110E';
   instHMIStationDriver.instsHSSPartSelect[3].lib.raw[5,7] := WSTRING#'16.32.112.315.017B';
   instHMIStationDriver.instsHSSPartSelect[3].lib.raw[6,0] := WSTRING#'';
   instHMIStationDriver.instsHSSPartSelect[3].lib.raw[6,1] := WSTRING#'C/O MATERIALS';
   instHMIStationDriver.instsHSSPartSelect[3].lib.raw[6,2] := WSTRING#'';
   instHMIStationDriver.instsHSSPartSelect[3].lib.raw[6,3] := WSTRING#'16.32.112.543.210E';
   instHMIStationDriver.instsHSSPartSelect[3].lib.raw[6,4] := WSTRING#'';
   instHMIStationDriver.instsHSSPartSelect[3].lib.raw[6,5] := WSTRING#'';
   instHMIStationDriver.instsHSSPartSelect[3].lib.raw[6,6] := WSTRING#'16.32.112.543.020A';
   instHMIStationDriver.instsHSSPartSelect[3].lib.raw[6,7] := WSTRING#'16.32.112.315.018A';
   instHMIStationDriver.instsHSSPartSelect[3].lib.raw[7,0] := WSTRING#'';
   instHMIStationDriver.instsHSSPartSelect[3].lib.raw[7,1] := WSTRING#'C/O MATERIALS';
   instHMIStationDriver.instsHSSPartSelect[3].lib.raw[7,2] := WSTRING#'16.08.216.291.000A';
   instHMIStationDriver.instsHSSPartSelect[3].lib.raw[7,3] := WSTRING#'16.08.216.315.001A';
   instHMIStationDriver.instsHSSPartSelect[3].lib.raw[7,4] := WSTRING#'';
   instHMIStationDriver.instsHSSPartSelect[3].lib.raw[7,5] := WSTRING#'16.08.216.057.001A';
   instHMIStationDriver.instsHSSPartSelect[3].lib.raw[7,6] := WSTRING#'16.08.208.661.000F';
   instHMIStationDriver.instsHSSPartSelect[3].lib.raw[7,7] := WSTRING#'16.08.216.315.002A';
   instHMIStationDriver.instsHSSPartSelect[3].lib.raw[8,0] := WSTRING#'';
   instHMIStationDriver.instsHSSPartSelect[3].lib.raw[8,1] := WSTRING#'C/O MATERIALS';
   instHMIStationDriver.instsHSSPartSelect[3].lib.raw[8,2] := WSTRING#'16.08.208.041.000A';
   instHMIStationDriver.instsHSSPartSelect[3].lib.raw[8,3] := WSTRING#'16.08.208.031.020C';
   instHMIStationDriver.instsHSSPartSelect[3].lib.raw[8,4] := WSTRING#'';
   instHMIStationDriver.instsHSSPartSelect[3].lib.raw[8,5] := WSTRING#'16.08.211.291.000A';
   instHMIStationDriver.instsHSSPartSelect[3].lib.raw[8,6] := WSTRING#'16.08.208.661.000F';
   instHMIStationDriver.instsHSSPartSelect[3].lib.raw[8,7] := WSTRING#'16.08.208.651.010B';
   instHMIStationDriver.instsHSSPartSelect[3].lib.raw[9,0] := WSTRING#'';
   instHMIStationDriver.instsHSSPartSelect[3].lib.raw[9,1] := WSTRING#'C/O MATERIALS';
   instHMIStationDriver.instsHSSPartSelect[3].lib.raw[9,2] := WSTRING#'16.08.211.806.020A';
   instHMIStationDriver.instsHSSPartSelect[3].lib.raw[9,3] := WSTRING#'';
   instHMIStationDriver.instsHSSPartSelect[3].lib.raw[9,4] := WSTRING#'';
   instHMIStationDriver.instsHSSPartSelect[3].lib.raw[9,5] := WSTRING#'';
   instHMIStationDriver.instsHSSPartSelect[3].lib.raw[9,6] := WSTRING#'16.08.208.631.000F';
   instHMIStationDriver.instsHSSPartSelect[3].lib.raw[9,7] := WSTRING#'16.08.216.315.000A';
   instHMIStationDriver.instsHSSPartSelect[3].lib.raw[10,0] := WSTRING#'';
   instHMIStationDriver.instsHSSPartSelect[3].lib.raw[10,1] := WSTRING#'C/O MATERIALS';
   instHMIStationDriver.instsHSSPartSelect[3].lib.raw[10,2] := WSTRING#'16.08.216.806.020A';
   instHMIStationDriver.instsHSSPartSelect[3].lib.raw[10,3] := WSTRING#'';
   instHMIStationDriver.instsHSSPartSelect[3].lib.raw[10,4] := WSTRING#'';
   instHMIStationDriver.instsHSSPartSelect[3].lib.raw[10,5] := WSTRING#'';
   instHMIStationDriver.instsHSSPartSelect[3].lib.raw[10,6] := WSTRING#'16.08.208.631.000F';
   instHMIStationDriver.instsHSSPartSelect[3].lib.raw[10,7] := WSTRING#'16.08.216.315.000A';
   instHMIStationDriver.instsHSSPartSelect[3].lib.raw[11,0] := WSTRING#'';
   instHMIStationDriver.instsHSSPartSelect[3].lib.raw[11,1] := WSTRING#'';
   instHMIStationDriver.instsHSSPartSelect[3].lib.raw[11,2] := WSTRING#'';
   instHMIStationDriver.instsHSSPartSelect[3].lib.raw[11,3] := WSTRING#'';
   instHMIStationDriver.instsHSSPartSelect[3].lib.raw[11,4] := WSTRING#'';
   instHMIStationDriver.instsHSSPartSelect[3].lib.raw[11,5] := WSTRING#'';
   instHMIStationDriver.instsHSSPartSelect[3].lib.raw[11,6] := WSTRING#'';
   instHMIStationDriver.instsHSSPartSelect[3].lib.raw[11,7] := WSTRING#'';
   instHMIStationDriver.instsHSSPartSelect[3].lib.raw[12,0] := WSTRING#'';
   instHMIStationDriver.instsHSSPartSelect[3].lib.raw[12,1] := WSTRING#'';
   instHMIStationDriver.instsHSSPartSelect[3].lib.raw[12,2] := WSTRING#'';
   instHMIStationDriver.instsHSSPartSelect[3].lib.raw[12,3] := WSTRING#'';
   instHMIStationDriver.instsHSSPartSelect[3].lib.raw[12,4] := WSTRING#'';
   instHMIStationDriver.instsHSSPartSelect[3].lib.raw[12,5] := WSTRING#'';
   instHMIStationDriver.instsHSSPartSelect[3].lib.raw[12,6] := WSTRING#'';
   instHMIStationDriver.instsHSSPartSelect[3].lib.raw[12,7] := WSTRING#'';
   instHMIStationDriver.instsHSSPartSelect[3].lib.raw[13,0] := WSTRING#'';
   instHMIStationDriver.instsHSSPartSelect[3].lib.raw[13,1] := WSTRING#'';
   instHMIStationDriver.instsHSSPartSelect[3].lib.raw[13,2] := WSTRING#'';
   instHMIStationDriver.instsHSSPartSelect[3].lib.raw[13,3] := WSTRING#'';
   instHMIStationDriver.instsHSSPartSelect[3].lib.raw[13,4] := WSTRING#'';
   instHMIStationDriver.instsHSSPartSelect[3].lib.raw[13,5] := WSTRING#'';
   instHMIStationDriver.instsHSSPartSelect[3].lib.raw[13,6] := WSTRING#'';
   instHMIStationDriver.instsHSSPartSelect[3].lib.raw[13,7] := WSTRING#'';
   instHMIStationDriver.instsHSSPartSelect[3].lib.raw[14,0] := WSTRING#'';
   instHMIStationDriver.instsHSSPartSelect[3].lib.raw[14,1] := WSTRING#'';
   instHMIStationDriver.instsHSSPartSelect[3].lib.raw[14,2] := WSTRING#'';
   instHMIStationDriver.instsHSSPartSelect[3].lib.raw[14,3] := WSTRING#'';
   instHMIStationDriver.instsHSSPartSelect[3].lib.raw[14,4] := WSTRING#'';
   instHMIStationDriver.instsHSSPartSelect[3].lib.raw[14,5] := WSTRING#'';
   instHMIStationDriver.instsHSSPartSelect[3].lib.raw[14,6] := WSTRING#'';
   instHMIStationDriver.instsHSSPartSelect[3].lib.raw[14,7] := WSTRING#'';
   instHMIStationDriver.instsHSSPartSelect[3].lib.raw[15,0] := WSTRING#'';
   instHMIStationDriver.instsHSSPartSelect[3].lib.raw[15,1] := WSTRING#'';
   instHMIStationDriver.instsHSSPartSelect[3].lib.raw[15,2] := WSTRING#'';
   instHMIStationDriver.instsHSSPartSelect[3].lib.raw[15,3] := WSTRING#'';
   instHMIStationDriver.instsHSSPartSelect[3].lib.raw[15,4] := WSTRING#'';
   instHMIStationDriver.instsHSSPartSelect[3].lib.raw[15,5] := WSTRING#'';
   instHMIStationDriver.instsHSSPartSelect[3].lib.raw[15,6] := WSTRING#'';
   instHMIStationDriver.instsHSSPartSelect[3].lib.raw[15,7] := WSTRING#'';
   instHMIStationDriver.instsHSSPartSelect[3].lib.raw[16,0] := WSTRING#'';
   instHMIStationDriver.instsHSSPartSelect[3].lib.raw[16,1] := WSTRING#'';
   instHMIStationDriver.instsHSSPartSelect[3].lib.raw[16,2] := WSTRING#'';
   instHMIStationDriver.instsHSSPartSelect[3].lib.raw[16,3] := WSTRING#'';
   instHMIStationDriver.instsHSSPartSelect[3].lib.raw[16,4] := WSTRING#'';
   instHMIStationDriver.instsHSSPartSelect[3].lib.raw[16,5] := WSTRING#'';
   instHMIStationDriver.instsHSSPartSelect[3].lib.raw[16,6] := WSTRING#'';
   instHMIStationDriver.instsHSSPartSelect[3].lib.raw[16,7] := WSTRING#'';
   instHMIStationDriver.instsHSSPartSelect[3].lib.raw[17,0] := WSTRING#'';
   instHMIStationDriver.instsHSSPartSelect[3].lib.raw[17,1] := WSTRING#'';
   instHMIStationDriver.instsHSSPartSelect[3].lib.raw[17,2] := WSTRING#'';
   instHMIStationDriver.instsHSSPartSelect[3].lib.raw[17,3] := WSTRING#'';
   instHMIStationDriver.instsHSSPartSelect[3].lib.raw[17,4] := WSTRING#'';
   instHMIStationDriver.instsHSSPartSelect[3].lib.raw[17,5] := WSTRING#'';
   instHMIStationDriver.instsHSSPartSelect[3].lib.raw[17,6] := WSTRING#'';
   instHMIStationDriver.instsHSSPartSelect[3].lib.raw[17,7] := WSTRING#'';
   instHMIStationDriver.instsHSSPartSelect[3].lib.raw[18,0] := WSTRING#'';
   instHMIStationDriver.instsHSSPartSelect[3].lib.raw[18,1] := WSTRING#'';
   instHMIStationDriver.instsHSSPartSelect[3].lib.raw[18,2] := WSTRING#'';
   instHMIStationDriver.instsHSSPartSelect[3].lib.raw[18,3] := WSTRING#'';
   instHMIStationDriver.instsHSSPartSelect[3].lib.raw[18,4] := WSTRING#'';
   instHMIStationDriver.instsHSSPartSelect[3].lib.raw[18,5] := WSTRING#'';
   instHMIStationDriver.instsHSSPartSelect[3].lib.raw[18,6] := WSTRING#'';
   instHMIStationDriver.instsHSSPartSelect[3].lib.raw[18,7] := WSTRING#'';
   instHMIStationDriver.instsHSSPartSelect[3].lib.raw[19,0] := WSTRING#'';
   instHMIStationDriver.instsHSSPartSelect[3].lib.raw[19,1] := WSTRING#'';
   instHMIStationDriver.instsHSSPartSelect[3].lib.raw[19,2] := WSTRING#'';
   instHMIStationDriver.instsHSSPartSelect[3].lib.raw[19,3] := WSTRING#'';
   instHMIStationDriver.instsHSSPartSelect[3].lib.raw[19,4] := WSTRING#'';
   instHMIStationDriver.instsHSSPartSelect[3].lib.raw[19,5] := WSTRING#'';
   instHMIStationDriver.instsHSSPartSelect[3].lib.raw[19,6] := WSTRING#'';
   instHMIStationDriver.instsHSSPartSelect[3].lib.raw[19,7] := WSTRING#'';
   instHMIStationDriver.instsHSSPartSelect[3].lib.raw[20,0] := WSTRING#'';
   instHMIStationDriver.instsHSSPartSelect[3].lib.raw[20,1] := WSTRING#'';
   instHMIStationDriver.instsHSSPartSelect[3].lib.raw[20,2] := WSTRING#'';
   instHMIStationDriver.instsHSSPartSelect[3].lib.raw[20,3] := WSTRING#'';
   instHMIStationDriver.instsHSSPartSelect[3].lib.raw[20,4] := WSTRING#'';
   instHMIStationDriver.instsHSSPartSelect[3].lib.raw[20,5] := WSTRING#'';
   instHMIStationDriver.instsHSSPartSelect[3].lib.raw[20,6] := WSTRING#'';
   instHMIStationDriver.instsHSSPartSelect[3].lib.raw[20,7] := WSTRING#'';
   instHMIStationDriver.instsHSSPartSelect[3].lib.raw[21,0] := WSTRING#'';
   instHMIStationDriver.instsHSSPartSelect[3].lib.raw[21,1] := WSTRING#'';
   instHMIStationDriver.instsHSSPartSelect[3].lib.raw[21,2] := WSTRING#'';
   instHMIStationDriver.instsHSSPartSelect[3].lib.raw[21,3] := WSTRING#'';
   instHMIStationDriver.instsHSSPartSelect[3].lib.raw[21,4] := WSTRING#'';
   instHMIStationDriver.instsHSSPartSelect[3].lib.raw[21,5] := WSTRING#'';
   instHMIStationDriver.instsHSSPartSelect[3].lib.raw[21,6] := WSTRING#'';
   instHMIStationDriver.instsHSSPartSelect[3].lib.raw[21,7] := WSTRING#'';
   instHMIStationDriver.instsHSSPartSelect[3].lib.raw[22,0] := WSTRING#'';
   instHMIStationDriver.instsHSSPartSelect[3].lib.raw[22,1] := WSTRING#'';
   instHMIStationDriver.instsHSSPartSelect[3].lib.raw[22,2] := WSTRING#'';
   instHMIStationDriver.instsHSSPartSelect[3].lib.raw[22,3] := WSTRING#'';
   instHMIStationDriver.instsHSSPartSelect[3].lib.raw[22,4] := WSTRING#'';
   instHMIStationDriver.instsHSSPartSelect[3].lib.raw[22,5] := WSTRING#'';
   instHMIStationDriver.instsHSSPartSelect[3].lib.raw[22,6] := WSTRING#'';
   instHMIStationDriver.instsHSSPartSelect[3].lib.raw[22,7] := WSTRING#'';
   instHMIStationDriver.instsHSSPartSelect[3].lib.raw[23,0] := WSTRING#'';
   instHMIStationDriver.instsHSSPartSelect[3].lib.raw[23,1] := WSTRING#'';
   instHMIStationDriver.instsHSSPartSelect[3].lib.raw[23,2] := WSTRING#'';
   instHMIStationDriver.instsHSSPartSelect[3].lib.raw[23,3] := WSTRING#'';
   instHMIStationDriver.instsHSSPartSelect[3].lib.raw[23,4] := WSTRING#'';
   instHMIStationDriver.instsHSSPartSelect[3].lib.raw[23,5] := WSTRING#'';
   instHMIStationDriver.instsHSSPartSelect[3].lib.raw[23,6] := WSTRING#'';
   instHMIStationDriver.instsHSSPartSelect[3].lib.raw[23,7] := WSTRING#'';
   instHMIStationDriver.instsHSSPartSelect[3].lib.raw[24,0] := WSTRING#'';
   instHMIStationDriver.instsHSSPartSelect[3].lib.raw[24,1] := WSTRING#'';
   instHMIStationDriver.instsHSSPartSelect[3].lib.raw[24,2] := WSTRING#'';
   instHMIStationDriver.instsHSSPartSelect[3].lib.raw[24,3] := WSTRING#'';
   instHMIStationDriver.instsHSSPartSelect[3].lib.raw[24,4] := WSTRING#'';
   instHMIStationDriver.instsHSSPartSelect[3].lib.raw[24,5] := WSTRING#'';
   instHMIStationDriver.instsHSSPartSelect[3].lib.raw[24,6] := WSTRING#'';
   instHMIStationDriver.instsHSSPartSelect[3].lib.raw[24,7] := WSTRING#'';
   instHMIStationDriver.instsHSSPartSelect[3].lib.raw[25,0] := WSTRING#'';
   instHMIStationDriver.instsHSSPartSelect[3].lib.raw[25,1] := WSTRING#'';
   instHMIStationDriver.instsHSSPartSelect[3].lib.raw[25,2] := WSTRING#'';
   instHMIStationDriver.instsHSSPartSelect[3].lib.raw[25,3] := WSTRING#'';
   instHMIStationDriver.instsHSSPartSelect[3].lib.raw[25,4] := WSTRING#'';
   instHMIStationDriver.instsHSSPartSelect[3].lib.raw[25,5] := WSTRING#'';
   instHMIStationDriver.instsHSSPartSelect[3].lib.raw[25,6] := WSTRING#'';
   instHMIStationDriver.instsHSSPartSelect[3].lib.raw[25,7] := WSTRING#'';
   instHMIStationDriver.instsHSSPartSelect[3].lib.raw[26,0] := WSTRING#'';
   instHMIStationDriver.instsHSSPartSelect[3].lib.raw[26,1] := WSTRING#'';
   instHMIStationDriver.instsHSSPartSelect[3].lib.raw[26,2] := WSTRING#'';
   instHMIStationDriver.instsHSSPartSelect[3].lib.raw[26,3] := WSTRING#'';
   instHMIStationDriver.instsHSSPartSelect[3].lib.raw[26,4] := WSTRING#'';
   instHMIStationDriver.instsHSSPartSelect[3].lib.raw[26,5] := WSTRING#'';
   instHMIStationDriver.instsHSSPartSelect[3].lib.raw[26,6] := WSTRING#'';
   instHMIStationDriver.instsHSSPartSelect[3].lib.raw[26,7] := WSTRING#'';
   instHMIStationDriver.instsHSSPartSelect[3].lib.raw[27,0] := WSTRING#'';
   instHMIStationDriver.instsHSSPartSelect[3].lib.raw[27,1] := WSTRING#'';
   instHMIStationDriver.instsHSSPartSelect[3].lib.raw[27,2] := WSTRING#'';
   instHMIStationDriver.instsHSSPartSelect[3].lib.raw[27,3] := WSTRING#'';
   instHMIStationDriver.instsHSSPartSelect[3].lib.raw[27,4] := WSTRING#'';
   instHMIStationDriver.instsHSSPartSelect[3].lib.raw[27,5] := WSTRING#'';
   instHMIStationDriver.instsHSSPartSelect[3].lib.raw[27,6] := WSTRING#'';
   instHMIStationDriver.instsHSSPartSelect[3].lib.raw[27,7] := WSTRING#'';
   instHMIStationDriver.instsHSSPartSelect[3].lib.raw[28,0] := WSTRING#'';
   instHMIStationDriver.instsHSSPartSelect[3].lib.raw[28,1] := WSTRING#'';
   instHMIStationDriver.instsHSSPartSelect[3].lib.raw[28,2] := WSTRING#'';
   instHMIStationDriver.instsHSSPartSelect[3].lib.raw[28,3] := WSTRING#'';
   instHMIStationDriver.instsHSSPartSelect[3].lib.raw[28,4] := WSTRING#'';
   instHMIStationDriver.instsHSSPartSelect[3].lib.raw[28,5] := WSTRING#'';
   instHMIStationDriver.instsHSSPartSelect[3].lib.raw[28,6] := WSTRING#'';
   instHMIStationDriver.instsHSSPartSelect[3].lib.raw[28,7] := WSTRING#'';
   instHMIStationDriver.instsHSSPartSelect[3].lib.raw[29,0] := WSTRING#'';
   instHMIStationDriver.instsHSSPartSelect[3].lib.raw[29,1] := WSTRING#'';
   instHMIStationDriver.instsHSSPartSelect[3].lib.raw[29,2] := WSTRING#'';
   instHMIStationDriver.instsHSSPartSelect[3].lib.raw[29,3] := WSTRING#'';
   instHMIStationDriver.instsHSSPartSelect[3].lib.raw[29,4] := WSTRING#'';
   instHMIStationDriver.instsHSSPartSelect[3].lib.raw[29,5] := WSTRING#'';
   instHMIStationDriver.instsHSSPartSelect[3].lib.raw[29,6] := WSTRING#'';
   instHMIStationDriver.instsHSSPartSelect[3].lib.raw[29,7] := WSTRING#'';
   instHMIStationDriver.instsHSSPartSelect[3].lib.raw[30,0] := WSTRING#'';
   instHMIStationDriver.instsHSSPartSelect[3].lib.raw[30,1] := WSTRING#'';
   instHMIStationDriver.instsHSSPartSelect[3].lib.raw[30,2] := WSTRING#'';
   instHMIStationDriver.instsHSSPartSelect[3].lib.raw[30,3] := WSTRING#'';
   instHMIStationDriver.instsHSSPartSelect[3].lib.raw[30,4] := WSTRING#'';
   instHMIStationDriver.instsHSSPartSelect[3].lib.raw[30,5] := WSTRING#'';
   instHMIStationDriver.instsHSSPartSelect[3].lib.raw[30,6] := WSTRING#'';
   instHMIStationDriver.instsHSSPartSelect[3].lib.raw[30,7] := WSTRING#'';
   instHMIStationDriver.instsHSSPartSelect[3].lib.raw[31,0] := WSTRING#'';
   instHMIStationDriver.instsHSSPartSelect[3].lib.raw[31,1] := WSTRING#'';
   instHMIStationDriver.instsHSSPartSelect[3].lib.raw[31,2] := WSTRING#'';
   instHMIStationDriver.instsHSSPartSelect[3].lib.raw[31,3] := WSTRING#'';
   instHMIStationDriver.instsHSSPartSelect[3].lib.raw[31,4] := WSTRING#'';
   instHMIStationDriver.instsHSSPartSelect[3].lib.raw[31,5] := WSTRING#'';
   instHMIStationDriver.instsHSSPartSelect[3].lib.raw[31,6] := WSTRING#'';
   instHMIStationDriver.instsHSSPartSelect[3].lib.raw[31,7] := WSTRING#'';
   instHMIStationDriver.instsHSSPartSelect[3].lib.raw[32,0] := WSTRING#'';
   instHMIStationDriver.instsHSSPartSelect[3].lib.raw[32,1] := WSTRING#'';
   instHMIStationDriver.instsHSSPartSelect[3].lib.raw[32,2] := WSTRING#'';
   instHMIStationDriver.instsHSSPartSelect[3].lib.raw[32,3] := WSTRING#'';
   instHMIStationDriver.instsHSSPartSelect[3].lib.raw[32,4] := WSTRING#'';
   instHMIStationDriver.instsHSSPartSelect[3].lib.raw[32,5] := WSTRING#'';
   instHMIStationDriver.instsHSSPartSelect[3].lib.raw[32,6] := WSTRING#'';
   instHMIStationDriver.instsHSSPartSelect[3].lib.raw[32,7] := WSTRING#'';
   instHMIStationDriver.instsHSSPartSelect[3].lib.raw[33,0] := WSTRING#'';
   instHMIStationDriver.instsHSSPartSelect[3].lib.raw[33,1] := WSTRING#'';
   instHMIStationDriver.instsHSSPartSelect[3].lib.raw[33,2] := WSTRING#'';
   instHMIStationDriver.instsHSSPartSelect[3].lib.raw[33,3] := WSTRING#'';
   instHMIStationDriver.instsHSSPartSelect[3].lib.raw[33,4] := WSTRING#'';
   instHMIStationDriver.instsHSSPartSelect[3].lib.raw[33,5] := WSTRING#'';
   instHMIStationDriver.instsHSSPartSelect[3].lib.raw[33,6] := WSTRING#'';
   instHMIStationDriver.instsHSSPartSelect[3].lib.raw[33,7] := WSTRING#'';
   instHMIStationDriver.instsHSSPartSelect[3].lib.raw[34,0] := WSTRING#'';
   instHMIStationDriver.instsHSSPartSelect[3].lib.raw[34,1] := WSTRING#'';
   instHMIStationDriver.instsHSSPartSelect[3].lib.raw[34,2] := WSTRING#'';
   instHMIStationDriver.instsHSSPartSelect[3].lib.raw[34,3] := WSTRING#'';
   instHMIStationDriver.instsHSSPartSelect[3].lib.raw[34,4] := WSTRING#'';
   instHMIStationDriver.instsHSSPartSelect[3].lib.raw[34,5] := WSTRING#'';
   instHMIStationDriver.instsHSSPartSelect[3].lib.raw[34,6] := WSTRING#'';
   instHMIStationDriver.instsHSSPartSelect[3].lib.raw[34,7] := WSTRING#'';
   instHMIStationDriver.instsHSSPartSelect[3].lib.raw[35,0] := WSTRING#'';
   instHMIStationDriver.instsHSSPartSelect[3].lib.raw[35,1] := WSTRING#'';
   instHMIStationDriver.instsHSSPartSelect[3].lib.raw[35,2] := WSTRING#'';
   instHMIStationDriver.instsHSSPartSelect[3].lib.raw[35,3] := WSTRING#'';
   instHMIStationDriver.instsHSSPartSelect[3].lib.raw[35,4] := WSTRING#'';
   instHMIStationDriver.instsHSSPartSelect[3].lib.raw[35,5] := WSTRING#'';
   instHMIStationDriver.instsHSSPartSelect[3].lib.raw[35,6] := WSTRING#'';
   instHMIStationDriver.instsHSSPartSelect[3].lib.raw[35,7] := WSTRING#'';
   instHMIStationDriver.instsHSSPartSelect[3].lib.raw[36,0] := WSTRING#'';
   instHMIStationDriver.instsHSSPartSelect[3].lib.raw[36,1] := WSTRING#'';
   instHMIStationDriver.instsHSSPartSelect[3].lib.raw[36,2] := WSTRING#'';
   instHMIStationDriver.instsHSSPartSelect[3].lib.raw[36,3] := WSTRING#'';
   instHMIStationDriver.instsHSSPartSelect[3].lib.raw[36,4] := WSTRING#'';
   instHMIStationDriver.instsHSSPartSelect[3].lib.raw[36,5] := WSTRING#'';
   instHMIStationDriver.instsHSSPartSelect[3].lib.raw[36,6] := WSTRING#'';
   instHMIStationDriver.instsHSSPartSelect[3].lib.raw[36,7] := WSTRING#'';
   instHMIStationDriver.instsHSSPartSelect[3].lib.raw[37,0] := WSTRING#'';
   instHMIStationDriver.instsHSSPartSelect[3].lib.raw[37,1] := WSTRING#'';
   instHMIStationDriver.instsHSSPartSelect[3].lib.raw[37,2] := WSTRING#'';
   instHMIStationDriver.instsHSSPartSelect[3].lib.raw[37,3] := WSTRING#'';
   instHMIStationDriver.instsHSSPartSelect[3].lib.raw[37,4] := WSTRING#'';
   instHMIStationDriver.instsHSSPartSelect[3].lib.raw[37,5] := WSTRING#'';
   instHMIStationDriver.instsHSSPartSelect[3].lib.raw[37,6] := WSTRING#'';
   instHMIStationDriver.instsHSSPartSelect[3].lib.raw[37,7] := WSTRING#'';
   instHMIStationDriver.instsHSSPartSelect[3].lib.raw[38,0] := WSTRING#'';
   instHMIStationDriver.instsHSSPartSelect[3].lib.raw[38,1] := WSTRING#'';
   instHMIStationDriver.instsHSSPartSelect[3].lib.raw[38,2] := WSTRING#'';
   instHMIStationDriver.instsHSSPartSelect[3].lib.raw[38,3] := WSTRING#'';
   instHMIStationDriver.instsHSSPartSelect[3].lib.raw[38,4] := WSTRING#'';
   instHMIStationDriver.instsHSSPartSelect[3].lib.raw[38,5] := WSTRING#'';
   instHMIStationDriver.instsHSSPartSelect[3].lib.raw[38,6] := WSTRING#'';
   instHMIStationDriver.instsHSSPartSelect[3].lib.raw[38,7] := WSTRING#'';
   instHMIStationDriver.instsHSSPartSelect[3].lib.raw[39,0] := WSTRING#'';
   instHMIStationDriver.instsHSSPartSelect[3].lib.raw[39,1] := WSTRING#'';
   instHMIStationDriver.instsHSSPartSelect[3].lib.raw[39,2] := WSTRING#'';
   instHMIStationDriver.instsHSSPartSelect[3].lib.raw[39,3] := WSTRING#'';
   instHMIStationDriver.instsHSSPartSelect[3].lib.raw[39,4] := WSTRING#'';
   instHMIStationDriver.instsHSSPartSelect[3].lib.raw[39,5] := WSTRING#'';
   instHMIStationDriver.instsHSSPartSelect[3].lib.raw[39,6] := WSTRING#'';
   instHMIStationDriver.instsHSSPartSelect[3].lib.raw[39,7] := WSTRING#'';
   instHMIStationDriver.instsHSSPartSelect[3].lib.raw[40,0] := WSTRING#'';
   instHMIStationDriver.instsHSSPartSelect[3].lib.raw[40,1] := WSTRING#'';
   instHMIStationDriver.instsHSSPartSelect[3].lib.raw[40,2] := WSTRING#'';
   instHMIStationDriver.instsHSSPartSelect[3].lib.raw[40,3] := WSTRING#'';
   instHMIStationDriver.instsHSSPartSelect[3].lib.raw[40,4] := WSTRING#'';
   instHMIStationDriver.instsHSSPartSelect[3].lib.raw[40,5] := WSTRING#'';
   instHMIStationDriver.instsHSSPartSelect[3].lib.raw[40,6] := WSTRING#'';
   instHMIStationDriver.instsHSSPartSelect[3].lib.raw[40,7] := WSTRING#'';
   instHMIStationDriver.instsHSSPartSelect[3].lib.raw[41,0] := WSTRING#'';
   instHMIStationDriver.instsHSSPartSelect[3].lib.raw[41,1] := WSTRING#'';
   instHMIStationDriver.instsHSSPartSelect[3].lib.raw[41,2] := WSTRING#'';
   instHMIStationDriver.instsHSSPartSelect[3].lib.raw[41,3] := WSTRING#'';
   instHMIStationDriver.instsHSSPartSelect[3].lib.raw[41,4] := WSTRING#'';
   instHMIStationDriver.instsHSSPartSelect[3].lib.raw[41,5] := WSTRING#'';
   instHMIStationDriver.instsHSSPartSelect[3].lib.raw[41,6] := WSTRING#'';
   instHMIStationDriver.instsHSSPartSelect[3].lib.raw[41,7] := WSTRING#'';
   instHMIStationDriver.instsHSSPartSelect[3].lib.raw[42,0] := WSTRING#'';
   instHMIStationDriver.instsHSSPartSelect[3].lib.raw[42,1] := WSTRING#'';
   instHMIStationDriver.instsHSSPartSelect[3].lib.raw[42,2] := WSTRING#'';
   instHMIStationDriver.instsHSSPartSelect[3].lib.raw[42,3] := WSTRING#'';
   instHMIStationDriver.instsHSSPartSelect[3].lib.raw[42,4] := WSTRING#'';
   instHMIStationDriver.instsHSSPartSelect[3].lib.raw[42,5] := WSTRING#'';
   instHMIStationDriver.instsHSSPartSelect[3].lib.raw[42,6] := WSTRING#'';
   instHMIStationDriver.instsHSSPartSelect[3].lib.raw[42,7] := WSTRING#'';
   instHMIStationDriver.instsHSSPartSelect[3].lib.raw[43,0] := WSTRING#'';
   instHMIStationDriver.instsHSSPartSelect[3].lib.raw[43,1] := WSTRING#'';
   instHMIStationDriver.instsHSSPartSelect[3].lib.raw[43,2] := WSTRING#'';
   instHMIStationDriver.instsHSSPartSelect[3].lib.raw[43,3] := WSTRING#'';
   instHMIStationDriver.instsHSSPartSelect[3].lib.raw[43,4] := WSTRING#'';
   instHMIStationDriver.instsHSSPartSelect[3].lib.raw[43,5] := WSTRING#'';
   instHMIStationDriver.instsHSSPartSelect[3].lib.raw[43,6] := WSTRING#'';
   instHMIStationDriver.instsHSSPartSelect[3].lib.raw[43,7] := WSTRING#'';
   instHMIStationDriver.instsHSSPartSelect[3].lib.raw[44,0] := WSTRING#'';
   instHMIStationDriver.instsHSSPartSelect[3].lib.raw[44,1] := WSTRING#'';
   instHMIStationDriver.instsHSSPartSelect[3].lib.raw[44,2] := WSTRING#'';
   instHMIStationDriver.instsHSSPartSelect[3].lib.raw[44,3] := WSTRING#'';
   instHMIStationDriver.instsHSSPartSelect[3].lib.raw[44,4] := WSTRING#'';
   instHMIStationDriver.instsHSSPartSelect[3].lib.raw[44,5] := WSTRING#'';
   instHMIStationDriver.instsHSSPartSelect[3].lib.raw[44,6] := WSTRING#'';
   instHMIStationDriver.instsHSSPartSelect[3].lib.raw[44,7] := WSTRING#'';
   instHMIStationDriver.instsHSSPartSelect[3].lib.raw[45,0] := WSTRING#'';
   instHMIStationDriver.instsHSSPartSelect[3].lib.raw[45,1] := WSTRING#'';
   instHMIStationDriver.instsHSSPartSelect[3].lib.raw[45,2] := WSTRING#'';
   instHMIStationDriver.instsHSSPartSelect[3].lib.raw[45,3] := WSTRING#'';
   instHMIStationDriver.instsHSSPartSelect[3].lib.raw[45,4] := WSTRING#'';
   instHMIStationDriver.instsHSSPartSelect[3].lib.raw[45,5] := WSTRING#'';
   instHMIStationDriver.instsHSSPartSelect[3].lib.raw[45,6] := WSTRING#'';
   instHMIStationDriver.instsHSSPartSelect[3].lib.raw[45,7] := WSTRING#'';
   instHMIStationDriver.instsHSSPartSelect[3].lib.raw[46,0] := WSTRING#'';
   instHMIStationDriver.instsHSSPartSelect[3].lib.raw[46,1] := WSTRING#'';
   instHMIStationDriver.instsHSSPartSelect[3].lib.raw[46,2] := WSTRING#'';
   instHMIStationDriver.instsHSSPartSelect[3].lib.raw[46,3] := WSTRING#'';
   instHMIStationDriver.instsHSSPartSelect[3].lib.raw[46,4] := WSTRING#'';
   instHMIStationDriver.instsHSSPartSelect[3].lib.raw[46,5] := WSTRING#'';
   instHMIStationDriver.instsHSSPartSelect[3].lib.raw[46,6] := WSTRING#'';
   instHMIStationDriver.instsHSSPartSelect[3].lib.raw[46,7] := WSTRING#'';
   instHMIStationDriver.instsHSSPartSelect[3].lib.raw[47,0] := WSTRING#'';
   instHMIStationDriver.instsHSSPartSelect[3].lib.raw[47,1] := WSTRING#'';
   instHMIStationDriver.instsHSSPartSelect[3].lib.raw[47,2] := WSTRING#'';
   instHMIStationDriver.instsHSSPartSelect[3].lib.raw[47,3] := WSTRING#'';
   instHMIStationDriver.instsHSSPartSelect[3].lib.raw[47,4] := WSTRING#'';
   instHMIStationDriver.instsHSSPartSelect[3].lib.raw[47,5] := WSTRING#'';
   instHMIStationDriver.instsHSSPartSelect[3].lib.raw[47,6] := WSTRING#'';
   instHMIStationDriver.instsHSSPartSelect[3].lib.raw[47,7] := WSTRING#'';
   instHMIStationDriver.instsHSSPartSelect[3].lib.raw[48,0] := WSTRING#'';
   instHMIStationDriver.instsHSSPartSelect[3].lib.raw[48,1] := WSTRING#'';
   instHMIStationDriver.instsHSSPartSelect[3].lib.raw[48,2] := WSTRING#'';
   instHMIStationDriver.instsHSSPartSelect[3].lib.raw[48,3] := WSTRING#'';
   instHMIStationDriver.instsHSSPartSelect[3].lib.raw[48,4] := WSTRING#'';
   instHMIStationDriver.instsHSSPartSelect[3].lib.raw[48,5] := WSTRING#'';
   instHMIStationDriver.instsHSSPartSelect[3].lib.raw[48,6] := WSTRING#'';
   instHMIStationDriver.instsHSSPartSelect[3].lib.raw[48,7] := WSTRING#'';
   instHMIStationDriver.instsHSSPartSelect[3].lib.raw[49,0] := WSTRING#'';
   instHMIStationDriver.instsHSSPartSelect[3].lib.raw[49,1] := WSTRING#'';
   instHMIStationDriver.instsHSSPartSelect[3].lib.raw[49,2] := WSTRING#'';
   instHMIStationDriver.instsHSSPartSelect[3].lib.raw[49,3] := WSTRING#'';
   instHMIStationDriver.instsHSSPartSelect[3].lib.raw[49,4] := WSTRING#'';
   instHMIStationDriver.instsHSSPartSelect[3].lib.raw[49,5] := WSTRING#'';
   instHMIStationDriver.instsHSSPartSelect[3].lib.raw[49,6] := WSTRING#'';
   instHMIStationDriver.instsHSSPartSelect[3].lib.raw[49,7] := WSTRING#'';
   instHMIStationDriver.instsHSSPartSelect[4].recipeNum := 1;
   instHMIStationDriver.instsHSSPartSelect[4].lib.size := 3;
   instHMIStationDriver.instsHSSPartSelect[4].lib.wip[0] := WSTRING#'11.52.001.312.000B$LSA JL 2.2L DPF CANNING';
   instHMIStationDriver.instsHSSPartSelect[4].lib.wip[1] := WSTRING#'11.54.007.309.000D$LSTUFFED SHELL ASSEMBLY USA-U625';
   instHMIStationDriver.instsHSSPartSelect[4].lib.wip[2] := WSTRING#'11.54.007.309.002D$LSTUFFED SHELL ASSEMBLY USA-U625';
   instHMIStationDriver.instsHSSPartSelect[4].lib.wip[3] := WSTRING#'';
   instHMIStationDriver.instsHSSPartSelect[4].lib.wip[4] := WSTRING#'';
   instHMIStationDriver.instsHSSPartSelect[4].lib.wip[5] := WSTRING#'';
   instHMIStationDriver.instsHSSPartSelect[4].lib.wip[6] := WSTRING#'';
   instHMIStationDriver.instsHSSPartSelect[4].lib.wip[7] := WSTRING#'';
   instHMIStationDriver.instsHSSPartSelect[4].lib.wip[8] := WSTRING#'';
   instHMIStationDriver.instsHSSPartSelect[4].lib.wip[9] := WSTRING#'';
   instHMIStationDriver.instsHSSPartSelect[4].lib.wip[10] := WSTRING#'';
   instHMIStationDriver.instsHSSPartSelect[4].lib.wip[11] := WSTRING#'';
   instHMIStationDriver.instsHSSPartSelect[4].lib.wip[12] := WSTRING#'';
   instHMIStationDriver.instsHSSPartSelect[4].lib.wip[13] := WSTRING#'';
   instHMIStationDriver.instsHSSPartSelect[4].lib.wip[14] := WSTRING#'';
   instHMIStationDriver.instsHSSPartSelect[4].lib.wip[15] := WSTRING#'';
   instHMIStationDriver.instsHSSPartSelect[4].lib.wip[16] := WSTRING#'';
   instHMIStationDriver.instsHSSPartSelect[4].lib.wip[17] := WSTRING#'';
   instHMIStationDriver.instsHSSPartSelect[4].lib.wip[18] := WSTRING#'';
   instHMIStationDriver.instsHSSPartSelect[4].lib.wip[19] := WSTRING#'';
   instHMIStationDriver.instsHSSPartSelect[4].lib.wip[20] := WSTRING#'';
   instHMIStationDriver.instsHSSPartSelect[4].lib.wip[21] := WSTRING#'';
   instHMIStationDriver.instsHSSPartSelect[4].lib.wip[22] := WSTRING#'';
   instHMIStationDriver.instsHSSPartSelect[4].lib.wip[23] := WSTRING#'';
   instHMIStationDriver.instsHSSPartSelect[4].lib.wip[24] := WSTRING#'';
   instHMIStationDriver.instsHSSPartSelect[4].lib.wip[25] := WSTRING#'';
   instHMIStationDriver.instsHSSPartSelect[4].lib.wip[26] := WSTRING#'';
   instHMIStationDriver.instsHSSPartSelect[4].lib.wip[27] := WSTRING#'';
   instHMIStationDriver.instsHSSPartSelect[4].lib.wip[28] := WSTRING#'';
   instHMIStationDriver.instsHSSPartSelect[4].lib.wip[29] := WSTRING#'';
   instHMIStationDriver.instsHSSPartSelect[4].lib.wip[30] := WSTRING#'';
   instHMIStationDriver.instsHSSPartSelect[4].lib.wip[31] := WSTRING#'';
   instHMIStationDriver.instsHSSPartSelect[4].lib.wip[32] := WSTRING#'';
   instHMIStationDriver.instsHSSPartSelect[4].lib.wip[33] := WSTRING#'';
   instHMIStationDriver.instsHSSPartSelect[4].lib.wip[34] := WSTRING#'';
   instHMIStationDriver.instsHSSPartSelect[4].lib.wip[35] := WSTRING#'';
   instHMIStationDriver.instsHSSPartSelect[4].lib.wip[36] := WSTRING#'';
   instHMIStationDriver.instsHSSPartSelect[4].lib.wip[37] := WSTRING#'';
   instHMIStationDriver.instsHSSPartSelect[4].lib.wip[38] := WSTRING#'';
   instHMIStationDriver.instsHSSPartSelect[4].lib.wip[39] := WSTRING#'';
   instHMIStationDriver.instsHSSPartSelect[4].lib.wip[40] := WSTRING#'';
   instHMIStationDriver.instsHSSPartSelect[4].lib.wip[41] := WSTRING#'';
   instHMIStationDriver.instsHSSPartSelect[4].lib.wip[42] := WSTRING#'';
   instHMIStationDriver.instsHSSPartSelect[4].lib.wip[43] := WSTRING#'';
   instHMIStationDriver.instsHSSPartSelect[4].lib.wip[44] := WSTRING#'';
   instHMIStationDriver.instsHSSPartSelect[4].lib.wip[45] := WSTRING#'';
   instHMIStationDriver.instsHSSPartSelect[4].lib.wip[46] := WSTRING#'';
   instHMIStationDriver.instsHSSPartSelect[4].lib.wip[47] := WSTRING#'';
   instHMIStationDriver.instsHSSPartSelect[4].lib.wip[48] := WSTRING#'';
   instHMIStationDriver.instsHSSPartSelect[4].lib.wip[49] := WSTRING#'';
   instHMIStationDriver.instsHSSPartSelect[4].lib.raw[0,0] := WSTRING#'';
   instHMIStationDriver.instsHSSPartSelect[4].lib.raw[0,1] := WSTRING#'C/O MATERIALS';
   instHMIStationDriver.instsHSSPartSelect[4].lib.raw[0,2] := WSTRING#'';
   instHMIStationDriver.instsHSSPartSelect[4].lib.raw[0,3] := WSTRING#'11.52.001.316.001D';
   instHMIStationDriver.instsHSSPartSelect[4].lib.raw[0,4] := WSTRING#'';
   instHMIStationDriver.instsHSSPartSelect[4].lib.raw[0,5] := WSTRING#'';
   instHMIStationDriver.instsHSSPartSelect[4].lib.raw[0,6] := WSTRING#'11.52.001.055.000B';
   instHMIStationDriver.instsHSSPartSelect[4].lib.raw[0,7] := WSTRING#'11.52.001.315.000B';
   instHMIStationDriver.instsHSSPartSelect[4].lib.raw[1,0] := WSTRING#'';
   instHMIStationDriver.instsHSSPartSelect[4].lib.raw[1,1] := WSTRING#'C/O MATERIALS';
   instHMIStationDriver.instsHSSPartSelect[4].lib.raw[1,2] := WSTRING#'11.54.007.052.007B';
   instHMIStationDriver.instsHSSPartSelect[4].lib.raw[1,3] := WSTRING#'11.54.007.315.026G';
   instHMIStationDriver.instsHSSPartSelect[4].lib.raw[1,4] := WSTRING#'';
   instHMIStationDriver.instsHSSPartSelect[4].lib.raw[1,5] := WSTRING#'11.54.007.052.008A';
   instHMIStationDriver.instsHSSPartSelect[4].lib.raw[1,6] := WSTRING#'11.54.007.045.015D';
   instHMIStationDriver.instsHSSPartSelect[4].lib.raw[1,7] := WSTRING#'11.54.017.315.001F';
   instHMIStationDriver.instsHSSPartSelect[4].lib.raw[2,0] := WSTRING#'';
   instHMIStationDriver.instsHSSPartSelect[4].lib.raw[2,1] := WSTRING#'C/O MATERIALS';
   instHMIStationDriver.instsHSSPartSelect[4].lib.raw[2,2] := WSTRING#'11.54.007.052.009B';
   instHMIStationDriver.instsHSSPartSelect[4].lib.raw[2,3] := WSTRING#'11.54.007.315.026G';
   instHMIStationDriver.instsHSSPartSelect[4].lib.raw[2,4] := WSTRING#'';
   instHMIStationDriver.instsHSSPartSelect[4].lib.raw[2,5] := WSTRING#'11.54.007.052.010B';
   instHMIStationDriver.instsHSSPartSelect[4].lib.raw[2,6] := WSTRING#'11.54.007.045.015D';
   instHMIStationDriver.instsHSSPartSelect[4].lib.raw[2,7] := WSTRING#'11.54.017.315.001F';
   instHMIStationDriver.instsHSSPartSelect[4].lib.raw[3,0] := WSTRING#'';
   instHMIStationDriver.instsHSSPartSelect[4].lib.raw[3,1] := WSTRING#'';
   instHMIStationDriver.instsHSSPartSelect[4].lib.raw[3,2] := WSTRING#'';
   instHMIStationDriver.instsHSSPartSelect[4].lib.raw[3,3] := WSTRING#'';
   instHMIStationDriver.instsHSSPartSelect[4].lib.raw[3,4] := WSTRING#'';
   instHMIStationDriver.instsHSSPartSelect[4].lib.raw[3,5] := WSTRING#'';
   instHMIStationDriver.instsHSSPartSelect[4].lib.raw[3,6] := WSTRING#'';
   instHMIStationDriver.instsHSSPartSelect[4].lib.raw[3,7] := WSTRING#'';
   instHMIStationDriver.instsHSSPartSelect[4].lib.raw[4,0] := WSTRING#'';
   instHMIStationDriver.instsHSSPartSelect[4].lib.raw[4,1] := WSTRING#'';
   instHMIStationDriver.instsHSSPartSelect[4].lib.raw[4,2] := WSTRING#'';
   instHMIStationDriver.instsHSSPartSelect[4].lib.raw[4,3] := WSTRING#'';
   instHMIStationDriver.instsHSSPartSelect[4].lib.raw[4,4] := WSTRING#'';
   instHMIStationDriver.instsHSSPartSelect[4].lib.raw[4,5] := WSTRING#'';
   instHMIStationDriver.instsHSSPartSelect[4].lib.raw[4,6] := WSTRING#'';
   instHMIStationDriver.instsHSSPartSelect[4].lib.raw[4,7] := WSTRING#'';
   instHMIStationDriver.instsHSSPartSelect[4].lib.raw[5,0] := WSTRING#'';
   instHMIStationDriver.instsHSSPartSelect[4].lib.raw[5,1] := WSTRING#'';
   instHMIStationDriver.instsHSSPartSelect[4].lib.raw[5,2] := WSTRING#'';
   instHMIStationDriver.instsHSSPartSelect[4].lib.raw[5,3] := WSTRING#'';
   instHMIStationDriver.instsHSSPartSelect[4].lib.raw[5,4] := WSTRING#'';
   instHMIStationDriver.instsHSSPartSelect[4].lib.raw[5,5] := WSTRING#'';
   instHMIStationDriver.instsHSSPartSelect[4].lib.raw[5,6] := WSTRING#'';
   instHMIStationDriver.instsHSSPartSelect[4].lib.raw[5,7] := WSTRING#'';
   instHMIStationDriver.instsHSSPartSelect[4].lib.raw[6,0] := WSTRING#'';
   instHMIStationDriver.instsHSSPartSelect[4].lib.raw[6,1] := WSTRING#'';
   instHMIStationDriver.instsHSSPartSelect[4].lib.raw[6,2] := WSTRING#'';
   instHMIStationDriver.instsHSSPartSelect[4].lib.raw[6,3] := WSTRING#'';
   instHMIStationDriver.instsHSSPartSelect[4].lib.raw[6,4] := WSTRING#'';
   instHMIStationDriver.instsHSSPartSelect[4].lib.raw[6,5] := WSTRING#'';
   instHMIStationDriver.instsHSSPartSelect[4].lib.raw[6,6] := WSTRING#'';
   instHMIStationDriver.instsHSSPartSelect[4].lib.raw[6,7] := WSTRING#'';
   instHMIStationDriver.instsHSSPartSelect[4].lib.raw[7,0] := WSTRING#'';
   instHMIStationDriver.instsHSSPartSelect[4].lib.raw[7,1] := WSTRING#'';
   instHMIStationDriver.instsHSSPartSelect[4].lib.raw[7,2] := WSTRING#'';
   instHMIStationDriver.instsHSSPartSelect[4].lib.raw[7,3] := WSTRING#'';
   instHMIStationDriver.instsHSSPartSelect[4].lib.raw[7,4] := WSTRING#'';
   instHMIStationDriver.instsHSSPartSelect[4].lib.raw[7,5] := WSTRING#'';
   instHMIStationDriver.instsHSSPartSelect[4].lib.raw[7,6] := WSTRING#'';
   instHMIStationDriver.instsHSSPartSelect[4].lib.raw[7,7] := WSTRING#'';
   instHMIStationDriver.instsHSSPartSelect[4].lib.raw[8,0] := WSTRING#'';
   instHMIStationDriver.instsHSSPartSelect[4].lib.raw[8,1] := WSTRING#'';
   instHMIStationDriver.instsHSSPartSelect[4].lib.raw[8,2] := WSTRING#'';
   instHMIStationDriver.instsHSSPartSelect[4].lib.raw[8,3] := WSTRING#'';
   instHMIStationDriver.instsHSSPartSelect[4].lib.raw[8,4] := WSTRING#'';
   instHMIStationDriver.instsHSSPartSelect[4].lib.raw[8,5] := WSTRING#'';
   instHMIStationDriver.instsHSSPartSelect[4].lib.raw[8,6] := WSTRING#'';
   instHMIStationDriver.instsHSSPartSelect[4].lib.raw[8,7] := WSTRING#'';
   instHMIStationDriver.instsHSSPartSelect[4].lib.raw[9,0] := WSTRING#'';
   instHMIStationDriver.instsHSSPartSelect[4].lib.raw[9,1] := WSTRING#'';
   instHMIStationDriver.instsHSSPartSelect[4].lib.raw[9,2] := WSTRING#'';
   instHMIStationDriver.instsHSSPartSelect[4].lib.raw[9,3] := WSTRING#'';
   instHMIStationDriver.instsHSSPartSelect[4].lib.raw[9,4] := WSTRING#'';
   instHMIStationDriver.instsHSSPartSelect[4].lib.raw[9,5] := WSTRING#'';
   instHMIStationDriver.instsHSSPartSelect[4].lib.raw[9,6] := WSTRING#'';
   instHMIStationDriver.instsHSSPartSelect[4].lib.raw[9,7] := WSTRING#'';
   instHMIStationDriver.instsHSSPartSelect[4].lib.raw[10,0] := WSTRING#'';
   instHMIStationDriver.instsHSSPartSelect[4].lib.raw[10,1] := WSTRING#'';
   instHMIStationDriver.instsHSSPartSelect[4].lib.raw[10,2] := WSTRING#'';
   instHMIStationDriver.instsHSSPartSelect[4].lib.raw[10,3] := WSTRING#'';
   instHMIStationDriver.instsHSSPartSelect[4].lib.raw[10,4] := WSTRING#'';
   instHMIStationDriver.instsHSSPartSelect[4].lib.raw[10,5] := WSTRING#'';
   instHMIStationDriver.instsHSSPartSelect[4].lib.raw[10,6] := WSTRING#'';
   instHMIStationDriver.instsHSSPartSelect[4].lib.raw[10,7] := WSTRING#'';
   instHMIStationDriver.instsHSSPartSelect[4].lib.raw[11,0] := WSTRING#'';
   instHMIStationDriver.instsHSSPartSelect[4].lib.raw[11,1] := WSTRING#'';
   instHMIStationDriver.instsHSSPartSelect[4].lib.raw[11,2] := WSTRING#'';
   instHMIStationDriver.instsHSSPartSelect[4].lib.raw[11,3] := WSTRING#'';
   instHMIStationDriver.instsHSSPartSelect[4].lib.raw[11,4] := WSTRING#'';
   instHMIStationDriver.instsHSSPartSelect[4].lib.raw[11,5] := WSTRING#'';
   instHMIStationDriver.instsHSSPartSelect[4].lib.raw[11,6] := WSTRING#'';
   instHMIStationDriver.instsHSSPartSelect[4].lib.raw[11,7] := WSTRING#'';
   instHMIStationDriver.instsHSSPartSelect[4].lib.raw[12,0] := WSTRING#'';
   instHMIStationDriver.instsHSSPartSelect[4].lib.raw[12,1] := WSTRING#'';
   instHMIStationDriver.instsHSSPartSelect[4].lib.raw[12,2] := WSTRING#'';
   instHMIStationDriver.instsHSSPartSelect[4].lib.raw[12,3] := WSTRING#'';
   instHMIStationDriver.instsHSSPartSelect[4].lib.raw[12,4] := WSTRING#'';
   instHMIStationDriver.instsHSSPartSelect[4].lib.raw[12,5] := WSTRING#'';
   instHMIStationDriver.instsHSSPartSelect[4].lib.raw[12,6] := WSTRING#'';
   instHMIStationDriver.instsHSSPartSelect[4].lib.raw[12,7] := WSTRING#'';
   instHMIStationDriver.instsHSSPartSelect[4].lib.raw[13,0] := WSTRING#'';
   instHMIStationDriver.instsHSSPartSelect[4].lib.raw[13,1] := WSTRING#'';
   instHMIStationDriver.instsHSSPartSelect[4].lib.raw[13,2] := WSTRING#'';
   instHMIStationDriver.instsHSSPartSelect[4].lib.raw[13,3] := WSTRING#'';
   instHMIStationDriver.instsHSSPartSelect[4].lib.raw[13,4] := WSTRING#'';
   instHMIStationDriver.instsHSSPartSelect[4].lib.raw[13,5] := WSTRING#'';
   instHMIStationDriver.instsHSSPartSelect[4].lib.raw[13,6] := WSTRING#'';
   instHMIStationDriver.instsHSSPartSelect[4].lib.raw[13,7] := WSTRING#'';
   instHMIStationDriver.instsHSSPartSelect[4].lib.raw[14,0] := WSTRING#'';
   instHMIStationDriver.instsHSSPartSelect[4].lib.raw[14,1] := WSTRING#'';
   instHMIStationDriver.instsHSSPartSelect[4].lib.raw[14,2] := WSTRING#'';
   instHMIStationDriver.instsHSSPartSelect[4].lib.raw[14,3] := WSTRING#'';
   instHMIStationDriver.instsHSSPartSelect[4].lib.raw[14,4] := WSTRING#'';
   instHMIStationDriver.instsHSSPartSelect[4].lib.raw[14,5] := WSTRING#'';
   instHMIStationDriver.instsHSSPartSelect[4].lib.raw[14,6] := WSTRING#'';
   instHMIStationDriver.instsHSSPartSelect[4].lib.raw[14,7] := WSTRING#'';
   instHMIStationDriver.instsHSSPartSelect[4].lib.raw[15,0] := WSTRING#'';
   instHMIStationDriver.instsHSSPartSelect[4].lib.raw[15,1] := WSTRING#'';
   instHMIStationDriver.instsHSSPartSelect[4].lib.raw[15,2] := WSTRING#'';
   instHMIStationDriver.instsHSSPartSelect[4].lib.raw[15,3] := WSTRING#'';
   instHMIStationDriver.instsHSSPartSelect[4].lib.raw[15,4] := WSTRING#'';
   instHMIStationDriver.instsHSSPartSelect[4].lib.raw[15,5] := WSTRING#'';
   instHMIStationDriver.instsHSSPartSelect[4].lib.raw[15,6] := WSTRING#'';
   instHMIStationDriver.instsHSSPartSelect[4].lib.raw[15,7] := WSTRING#'';
   instHMIStationDriver.instsHSSPartSelect[4].lib.raw[16,0] := WSTRING#'';
   instHMIStationDriver.instsHSSPartSelect[4].lib.raw[16,1] := WSTRING#'';
   instHMIStationDriver.instsHSSPartSelect[4].lib.raw[16,2] := WSTRING#'';
   instHMIStationDriver.instsHSSPartSelect[4].lib.raw[16,3] := WSTRING#'';
   instHMIStationDriver.instsHSSPartSelect[4].lib.raw[16,4] := WSTRING#'';
   instHMIStationDriver.instsHSSPartSelect[4].lib.raw[16,5] := WSTRING#'';
   instHMIStationDriver.instsHSSPartSelect[4].lib.raw[16,6] := WSTRING#'';
   instHMIStationDriver.instsHSSPartSelect[4].lib.raw[16,7] := WSTRING#'';
   instHMIStationDriver.instsHSSPartSelect[4].lib.raw[17,0] := WSTRING#'';
   instHMIStationDriver.instsHSSPartSelect[4].lib.raw[17,1] := WSTRING#'';
   instHMIStationDriver.instsHSSPartSelect[4].lib.raw[17,2] := WSTRING#'';
   instHMIStationDriver.instsHSSPartSelect[4].lib.raw[17,3] := WSTRING#'';
   instHMIStationDriver.instsHSSPartSelect[4].lib.raw[17,4] := WSTRING#'';
   instHMIStationDriver.instsHSSPartSelect[4].lib.raw[17,5] := WSTRING#'';
   instHMIStationDriver.instsHSSPartSelect[4].lib.raw[17,6] := WSTRING#'';
   instHMIStationDriver.instsHSSPartSelect[4].lib.raw[17,7] := WSTRING#'';
   instHMIStationDriver.instsHSSPartSelect[4].lib.raw[18,0] := WSTRING#'';
   instHMIStationDriver.instsHSSPartSelect[4].lib.raw[18,1] := WSTRING#'';
   instHMIStationDriver.instsHSSPartSelect[4].lib.raw[18,2] := WSTRING#'';
   instHMIStationDriver.instsHSSPartSelect[4].lib.raw[18,3] := WSTRING#'';
   instHMIStationDriver.instsHSSPartSelect[4].lib.raw[18,4] := WSTRING#'';
   instHMIStationDriver.instsHSSPartSelect[4].lib.raw[18,5] := WSTRING#'';
   instHMIStationDriver.instsHSSPartSelect[4].lib.raw[18,6] := WSTRING#'';
   instHMIStationDriver.instsHSSPartSelect[4].lib.raw[18,7] := WSTRING#'';
   instHMIStationDriver.instsHSSPartSelect[4].lib.raw[19,0] := WSTRING#'';
   instHMIStationDriver.instsHSSPartSelect[4].lib.raw[19,1] := WSTRING#'';
   instHMIStationDriver.instsHSSPartSelect[4].lib.raw[19,2] := WSTRING#'';
   instHMIStationDriver.instsHSSPartSelect[4].lib.raw[19,3] := WSTRING#'';
   instHMIStationDriver.instsHSSPartSelect[4].lib.raw[19,4] := WSTRING#'';
   instHMIStationDriver.instsHSSPartSelect[4].lib.raw[19,5] := WSTRING#'';
   instHMIStationDriver.instsHSSPartSelect[4].lib.raw[19,6] := WSTRING#'';
   instHMIStationDriver.instsHSSPartSelect[4].lib.raw[19,7] := WSTRING#'';
   instHMIStationDriver.instsHSSPartSelect[4].lib.raw[20,0] := WSTRING#'';
   instHMIStationDriver.instsHSSPartSelect[4].lib.raw[20,1] := WSTRING#'';
   instHMIStationDriver.instsHSSPartSelect[4].lib.raw[20,2] := WSTRING#'';
   instHMIStationDriver.instsHSSPartSelect[4].lib.raw[20,3] := WSTRING#'';
   instHMIStationDriver.instsHSSPartSelect[4].lib.raw[20,4] := WSTRING#'';
   instHMIStationDriver.instsHSSPartSelect[4].lib.raw[20,5] := WSTRING#'';
   instHMIStationDriver.instsHSSPartSelect[4].lib.raw[20,6] := WSTRING#'';
   instHMIStationDriver.instsHSSPartSelect[4].lib.raw[20,7] := WSTRING#'';
   instHMIStationDriver.instsHSSPartSelect[4].lib.raw[21,0] := WSTRING#'';
   instHMIStationDriver.instsHSSPartSelect[4].lib.raw[21,1] := WSTRING#'';
   instHMIStationDriver.instsHSSPartSelect[4].lib.raw[21,2] := WSTRING#'';
   instHMIStationDriver.instsHSSPartSelect[4].lib.raw[21,3] := WSTRING#'';
   instHMIStationDriver.instsHSSPartSelect[4].lib.raw[21,4] := WSTRING#'';
   instHMIStationDriver.instsHSSPartSelect[4].lib.raw[21,5] := WSTRING#'';
   instHMIStationDriver.instsHSSPartSelect[4].lib.raw[21,6] := WSTRING#'';
   instHMIStationDriver.instsHSSPartSelect[4].lib.raw[21,7] := WSTRING#'';
   instHMIStationDriver.instsHSSPartSelect[4].lib.raw[22,0] := WSTRING#'';
   instHMIStationDriver.instsHSSPartSelect[4].lib.raw[22,1] := WSTRING#'';
   instHMIStationDriver.instsHSSPartSelect[4].lib.raw[22,2] := WSTRING#'';
   instHMIStationDriver.instsHSSPartSelect[4].lib.raw[22,3] := WSTRING#'';
   instHMIStationDriver.instsHSSPartSelect[4].lib.raw[22,4] := WSTRING#'';
   instHMIStationDriver.instsHSSPartSelect[4].lib.raw[22,5] := WSTRING#'';
   instHMIStationDriver.instsHSSPartSelect[4].lib.raw[22,6] := WSTRING#'';
   instHMIStationDriver.instsHSSPartSelect[4].lib.raw[22,7] := WSTRING#'';
   instHMIStationDriver.instsHSSPartSelect[4].lib.raw[23,0] := WSTRING#'';
   instHMIStationDriver.instsHSSPartSelect[4].lib.raw[23,1] := WSTRING#'';
   instHMIStationDriver.instsHSSPartSelect[4].lib.raw[23,2] := WSTRING#'';
   instHMIStationDriver.instsHSSPartSelect[4].lib.raw[23,3] := WSTRING#'';
   instHMIStationDriver.instsHSSPartSelect[4].lib.raw[23,4] := WSTRING#'';
   instHMIStationDriver.instsHSSPartSelect[4].lib.raw[23,5] := WSTRING#'';
   instHMIStationDriver.instsHSSPartSelect[4].lib.raw[23,6] := WSTRING#'';
   instHMIStationDriver.instsHSSPartSelect[4].lib.raw[23,7] := WSTRING#'';
   instHMIStationDriver.instsHSSPartSelect[4].lib.raw[24,0] := WSTRING#'';
   instHMIStationDriver.instsHSSPartSelect[4].lib.raw[24,1] := WSTRING#'';
   instHMIStationDriver.instsHSSPartSelect[4].lib.raw[24,2] := WSTRING#'';
   instHMIStationDriver.instsHSSPartSelect[4].lib.raw[24,3] := WSTRING#'';
   instHMIStationDriver.instsHSSPartSelect[4].lib.raw[24,4] := WSTRING#'';
   instHMIStationDriver.instsHSSPartSelect[4].lib.raw[24,5] := WSTRING#'';
   instHMIStationDriver.instsHSSPartSelect[4].lib.raw[24,6] := WSTRING#'';
   instHMIStationDriver.instsHSSPartSelect[4].lib.raw[24,7] := WSTRING#'';
   instHMIStationDriver.instsHSSPartSelect[4].lib.raw[25,0] := WSTRING#'';
   instHMIStationDriver.instsHSSPartSelect[4].lib.raw[25,1] := WSTRING#'';
   instHMIStationDriver.instsHSSPartSelect[4].lib.raw[25,2] := WSTRING#'';
   instHMIStationDriver.instsHSSPartSelect[4].lib.raw[25,3] := WSTRING#'';
   instHMIStationDriver.instsHSSPartSelect[4].lib.raw[25,4] := WSTRING#'';
   instHMIStationDriver.instsHSSPartSelect[4].lib.raw[25,5] := WSTRING#'';
   instHMIStationDriver.instsHSSPartSelect[4].lib.raw[25,6] := WSTRING#'';
   instHMIStationDriver.instsHSSPartSelect[4].lib.raw[25,7] := WSTRING#'';
   instHMIStationDriver.instsHSSPartSelect[4].lib.raw[26,0] := WSTRING#'';
   instHMIStationDriver.instsHSSPartSelect[4].lib.raw[26,1] := WSTRING#'';
   instHMIStationDriver.instsHSSPartSelect[4].lib.raw[26,2] := WSTRING#'';
   instHMIStationDriver.instsHSSPartSelect[4].lib.raw[26,3] := WSTRING#'';
   instHMIStationDriver.instsHSSPartSelect[4].lib.raw[26,4] := WSTRING#'';
   instHMIStationDriver.instsHSSPartSelect[4].lib.raw[26,5] := WSTRING#'';
   instHMIStationDriver.instsHSSPartSelect[4].lib.raw[26,6] := WSTRING#'';
   instHMIStationDriver.instsHSSPartSelect[4].lib.raw[26,7] := WSTRING#'';
   instHMIStationDriver.instsHSSPartSelect[4].lib.raw[27,0] := WSTRING#'';
   instHMIStationDriver.instsHSSPartSelect[4].lib.raw[27,1] := WSTRING#'';
   instHMIStationDriver.instsHSSPartSelect[4].lib.raw[27,2] := WSTRING#'';
   instHMIStationDriver.instsHSSPartSelect[4].lib.raw[27,3] := WSTRING#'';
   instHMIStationDriver.instsHSSPartSelect[4].lib.raw[27,4] := WSTRING#'';
   instHMIStationDriver.instsHSSPartSelect[4].lib.raw[27,5] := WSTRING#'';
   instHMIStationDriver.instsHSSPartSelect[4].lib.raw[27,6] := WSTRING#'';
   instHMIStationDriver.instsHSSPartSelect[4].lib.raw[27,7] := WSTRING#'';
   instHMIStationDriver.instsHSSPartSelect[4].lib.raw[28,0] := WSTRING#'';
   instHMIStationDriver.instsHSSPartSelect[4].lib.raw[28,1] := WSTRING#'';
   instHMIStationDriver.instsHSSPartSelect[4].lib.raw[28,2] := WSTRING#'';
   instHMIStationDriver.instsHSSPartSelect[4].lib.raw[28,3] := WSTRING#'';
   instHMIStationDriver.instsHSSPartSelect[4].lib.raw[28,4] := WSTRING#'';
   instHMIStationDriver.instsHSSPartSelect[4].lib.raw[28,5] := WSTRING#'';
   instHMIStationDriver.instsHSSPartSelect[4].lib.raw[28,6] := WSTRING#'';
   instHMIStationDriver.instsHSSPartSelect[4].lib.raw[28,7] := WSTRING#'';
   instHMIStationDriver.instsHSSPartSelect[4].lib.raw[29,0] := WSTRING#'';
   instHMIStationDriver.instsHSSPartSelect[4].lib.raw[29,1] := WSTRING#'';
   instHMIStationDriver.instsHSSPartSelect[4].lib.raw[29,2] := WSTRING#'';
   instHMIStationDriver.instsHSSPartSelect[4].lib.raw[29,3] := WSTRING#'';
   instHMIStationDriver.instsHSSPartSelect[4].lib.raw[29,4] := WSTRING#'';
   instHMIStationDriver.instsHSSPartSelect[4].lib.raw[29,5] := WSTRING#'';
   instHMIStationDriver.instsHSSPartSelect[4].lib.raw[29,6] := WSTRING#'';
   instHMIStationDriver.instsHSSPartSelect[4].lib.raw[29,7] := WSTRING#'';
   instHMIStationDriver.instsHSSPartSelect[4].lib.raw[30,0] := WSTRING#'';
   instHMIStationDriver.instsHSSPartSelect[4].lib.raw[30,1] := WSTRING#'';
   instHMIStationDriver.instsHSSPartSelect[4].lib.raw[30,2] := WSTRING#'';
   instHMIStationDriver.instsHSSPartSelect[4].lib.raw[30,3] := WSTRING#'';
   instHMIStationDriver.instsHSSPartSelect[4].lib.raw[30,4] := WSTRING#'';
   instHMIStationDriver.instsHSSPartSelect[4].lib.raw[30,5] := WSTRING#'';
   instHMIStationDriver.instsHSSPartSelect[4].lib.raw[30,6] := WSTRING#'';
   instHMIStationDriver.instsHSSPartSelect[4].lib.raw[30,7] := WSTRING#'';
   instHMIStationDriver.instsHSSPartSelect[4].lib.raw[31,0] := WSTRING#'';
   instHMIStationDriver.instsHSSPartSelect[4].lib.raw[31,1] := WSTRING#'';
   instHMIStationDriver.instsHSSPartSelect[4].lib.raw[31,2] := WSTRING#'';
   instHMIStationDriver.instsHSSPartSelect[4].lib.raw[31,3] := WSTRING#'';
   instHMIStationDriver.instsHSSPartSelect[4].lib.raw[31,4] := WSTRING#'';
   instHMIStationDriver.instsHSSPartSelect[4].lib.raw[31,5] := WSTRING#'';
   instHMIStationDriver.instsHSSPartSelect[4].lib.raw[31,6] := WSTRING#'';
   instHMIStationDriver.instsHSSPartSelect[4].lib.raw[31,7] := WSTRING#'';
   instHMIStationDriver.instsHSSPartSelect[4].lib.raw[32,0] := WSTRING#'';
   instHMIStationDriver.instsHSSPartSelect[4].lib.raw[32,1] := WSTRING#'';
   instHMIStationDriver.instsHSSPartSelect[4].lib.raw[32,2] := WSTRING#'';
   instHMIStationDriver.instsHSSPartSelect[4].lib.raw[32,3] := WSTRING#'';
   instHMIStationDriver.instsHSSPartSelect[4].lib.raw[32,4] := WSTRING#'';
   instHMIStationDriver.instsHSSPartSelect[4].lib.raw[32,5] := WSTRING#'';
   instHMIStationDriver.instsHSSPartSelect[4].lib.raw[32,6] := WSTRING#'';
   instHMIStationDriver.instsHSSPartSelect[4].lib.raw[32,7] := WSTRING#'';
   instHMIStationDriver.instsHSSPartSelect[4].lib.raw[33,0] := WSTRING#'';
   instHMIStationDriver.instsHSSPartSelect[4].lib.raw[33,1] := WSTRING#'';
   instHMIStationDriver.instsHSSPartSelect[4].lib.raw[33,2] := WSTRING#'';
   instHMIStationDriver.instsHSSPartSelect[4].lib.raw[33,3] := WSTRING#'';
   instHMIStationDriver.instsHSSPartSelect[4].lib.raw[33,4] := WSTRING#'';
   instHMIStationDriver.instsHSSPartSelect[4].lib.raw[33,5] := WSTRING#'';
   instHMIStationDriver.instsHSSPartSelect[4].lib.raw[33,6] := WSTRING#'';
   instHMIStationDriver.instsHSSPartSelect[4].lib.raw[33,7] := WSTRING#'';
   instHMIStationDriver.instsHSSPartSelect[4].lib.raw[34,0] := WSTRING#'';
   instHMIStationDriver.instsHSSPartSelect[4].lib.raw[34,1] := WSTRING#'';
   instHMIStationDriver.instsHSSPartSelect[4].lib.raw[34,2] := WSTRING#'';
   instHMIStationDriver.instsHSSPartSelect[4].lib.raw[34,3] := WSTRING#'';
   instHMIStationDriver.instsHSSPartSelect[4].lib.raw[34,4] := WSTRING#'';
   instHMIStationDriver.instsHSSPartSelect[4].lib.raw[34,5] := WSTRING#'';
   instHMIStationDriver.instsHSSPartSelect[4].lib.raw[34,6] := WSTRING#'';
   instHMIStationDriver.instsHSSPartSelect[4].lib.raw[34,7] := WSTRING#'';
   instHMIStationDriver.instsHSSPartSelect[4].lib.raw[35,0] := WSTRING#'';
   instHMIStationDriver.instsHSSPartSelect[4].lib.raw[35,1] := WSTRING#'';
   instHMIStationDriver.instsHSSPartSelect[4].lib.raw[35,2] := WSTRING#'';
   instHMIStationDriver.instsHSSPartSelect[4].lib.raw[35,3] := WSTRING#'';
   instHMIStationDriver.instsHSSPartSelect[4].lib.raw[35,4] := WSTRING#'';
   instHMIStationDriver.instsHSSPartSelect[4].lib.raw[35,5] := WSTRING#'';
   instHMIStationDriver.instsHSSPartSelect[4].lib.raw[35,6] := WSTRING#'';
   instHMIStationDriver.instsHSSPartSelect[4].lib.raw[35,7] := WSTRING#'';
   instHMIStationDriver.instsHSSPartSelect[4].lib.raw[36,0] := WSTRING#'';
   instHMIStationDriver.instsHSSPartSelect[4].lib.raw[36,1] := WSTRING#'';
   instHMIStationDriver.instsHSSPartSelect[4].lib.raw[36,2] := WSTRING#'';
   instHMIStationDriver.instsHSSPartSelect[4].lib.raw[36,3] := WSTRING#'';
   instHMIStationDriver.instsHSSPartSelect[4].lib.raw[36,4] := WSTRING#'';
   instHMIStationDriver.instsHSSPartSelect[4].lib.raw[36,5] := WSTRING#'';
   instHMIStationDriver.instsHSSPartSelect[4].lib.raw[36,6] := WSTRING#'';
   instHMIStationDriver.instsHSSPartSelect[4].lib.raw[36,7] := WSTRING#'';
   instHMIStationDriver.instsHSSPartSelect[4].lib.raw[37,0] := WSTRING#'';
   instHMIStationDriver.instsHSSPartSelect[4].lib.raw[37,1] := WSTRING#'';
   instHMIStationDriver.instsHSSPartSelect[4].lib.raw[37,2] := WSTRING#'';
   instHMIStationDriver.instsHSSPartSelect[4].lib.raw[37,3] := WSTRING#'';
   instHMIStationDriver.instsHSSPartSelect[4].lib.raw[37,4] := WSTRING#'';
   instHMIStationDriver.instsHSSPartSelect[4].lib.raw[37,5] := WSTRING#'';
   instHMIStationDriver.instsHSSPartSelect[4].lib.raw[37,6] := WSTRING#'';
   instHMIStationDriver.instsHSSPartSelect[4].lib.raw[37,7] := WSTRING#'';
   instHMIStationDriver.instsHSSPartSelect[4].lib.raw[38,0] := WSTRING#'';
   instHMIStationDriver.instsHSSPartSelect[4].lib.raw[38,1] := WSTRING#'';
   instHMIStationDriver.instsHSSPartSelect[4].lib.raw[38,2] := WSTRING#'';
   instHMIStationDriver.instsHSSPartSelect[4].lib.raw[38,3] := WSTRING#'';
   instHMIStationDriver.instsHSSPartSelect[4].lib.raw[38,4] := WSTRING#'';
   instHMIStationDriver.instsHSSPartSelect[4].lib.raw[38,5] := WSTRING#'';
   instHMIStationDriver.instsHSSPartSelect[4].lib.raw[38,6] := WSTRING#'';
   instHMIStationDriver.instsHSSPartSelect[4].lib.raw[38,7] := WSTRING#'';
   instHMIStationDriver.instsHSSPartSelect[4].lib.raw[39,0] := WSTRING#'';
   instHMIStationDriver.instsHSSPartSelect[4].lib.raw[39,1] := WSTRING#'';
   instHMIStationDriver.instsHSSPartSelect[4].lib.raw[39,2] := WSTRING#'';
   instHMIStationDriver.instsHSSPartSelect[4].lib.raw[39,3] := WSTRING#'';
   instHMIStationDriver.instsHSSPartSelect[4].lib.raw[39,4] := WSTRING#'';
   instHMIStationDriver.instsHSSPartSelect[4].lib.raw[39,5] := WSTRING#'';
   instHMIStationDriver.instsHSSPartSelect[4].lib.raw[39,6] := WSTRING#'';
   instHMIStationDriver.instsHSSPartSelect[4].lib.raw[39,7] := WSTRING#'';
   instHMIStationDriver.instsHSSPartSelect[4].lib.raw[40,0] := WSTRING#'';
   instHMIStationDriver.instsHSSPartSelect[4].lib.raw[40,1] := WSTRING#'';
   instHMIStationDriver.instsHSSPartSelect[4].lib.raw[40,2] := WSTRING#'';
   instHMIStationDriver.instsHSSPartSelect[4].lib.raw[40,3] := WSTRING#'';
   instHMIStationDriver.instsHSSPartSelect[4].lib.raw[40,4] := WSTRING#'';
   instHMIStationDriver.instsHSSPartSelect[4].lib.raw[40,5] := WSTRING#'';
   instHMIStationDriver.instsHSSPartSelect[4].lib.raw[40,6] := WSTRING#'';
   instHMIStationDriver.instsHSSPartSelect[4].lib.raw[40,7] := WSTRING#'';
   instHMIStationDriver.instsHSSPartSelect[4].lib.raw[41,0] := WSTRING#'';
   instHMIStationDriver.instsHSSPartSelect[4].lib.raw[41,1] := WSTRING#'';
   instHMIStationDriver.instsHSSPartSelect[4].lib.raw[41,2] := WSTRING#'';
   instHMIStationDriver.instsHSSPartSelect[4].lib.raw[41,3] := WSTRING#'';
   instHMIStationDriver.instsHSSPartSelect[4].lib.raw[41,4] := WSTRING#'';
   instHMIStationDriver.instsHSSPartSelect[4].lib.raw[41,5] := WSTRING#'';
   instHMIStationDriver.instsHSSPartSelect[4].lib.raw[41,6] := WSTRING#'';
   instHMIStationDriver.instsHSSPartSelect[4].lib.raw[41,7] := WSTRING#'';
   instHMIStationDriver.instsHSSPartSelect[4].lib.raw[42,0] := WSTRING#'';
   instHMIStationDriver.instsHSSPartSelect[4].lib.raw[42,1] := WSTRING#'';
   instHMIStationDriver.instsHSSPartSelect[4].lib.raw[42,2] := WSTRING#'';
   instHMIStationDriver.instsHSSPartSelect[4].lib.raw[42,3] := WSTRING#'';
   instHMIStationDriver.instsHSSPartSelect[4].lib.raw[42,4] := WSTRING#'';
   instHMIStationDriver.instsHSSPartSelect[4].lib.raw[42,5] := WSTRING#'';
   instHMIStationDriver.instsHSSPartSelect[4].lib.raw[42,6] := WSTRING#'';
   instHMIStationDriver.instsHSSPartSelect[4].lib.raw[42,7] := WSTRING#'';
   instHMIStationDriver.instsHSSPartSelect[4].lib.raw[43,0] := WSTRING#'';
   instHMIStationDriver.instsHSSPartSelect[4].lib.raw[43,1] := WSTRING#'';
   instHMIStationDriver.instsHSSPartSelect[4].lib.raw[43,2] := WSTRING#'';
   instHMIStationDriver.instsHSSPartSelect[4].lib.raw[43,3] := WSTRING#'';
   instHMIStationDriver.instsHSSPartSelect[4].lib.raw[43,4] := WSTRING#'';
   instHMIStationDriver.instsHSSPartSelect[4].lib.raw[43,5] := WSTRING#'';
   instHMIStationDriver.instsHSSPartSelect[4].lib.raw[43,6] := WSTRING#'';
   instHMIStationDriver.instsHSSPartSelect[4].lib.raw[43,7] := WSTRING#'';
   instHMIStationDriver.instsHSSPartSelect[4].lib.raw[44,0] := WSTRING#'';
   instHMIStationDriver.instsHSSPartSelect[4].lib.raw[44,1] := WSTRING#'';
   instHMIStationDriver.instsHSSPartSelect[4].lib.raw[44,2] := WSTRING#'';
   instHMIStationDriver.instsHSSPartSelect[4].lib.raw[44,3] := WSTRING#'';
   instHMIStationDriver.instsHSSPartSelect[4].lib.raw[44,4] := WSTRING#'';
   instHMIStationDriver.instsHSSPartSelect[4].lib.raw[44,5] := WSTRING#'';
   instHMIStationDriver.instsHSSPartSelect[4].lib.raw[44,6] := WSTRING#'';
   instHMIStationDriver.instsHSSPartSelect[4].lib.raw[44,7] := WSTRING#'';
   instHMIStationDriver.instsHSSPartSelect[4].lib.raw[45,0] := WSTRING#'';
   instHMIStationDriver.instsHSSPartSelect[4].lib.raw[45,1] := WSTRING#'';
   instHMIStationDriver.instsHSSPartSelect[4].lib.raw[45,2] := WSTRING#'';
   instHMIStationDriver.instsHSSPartSelect[4].lib.raw[45,3] := WSTRING#'';
   instHMIStationDriver.instsHSSPartSelect[4].lib.raw[45,4] := WSTRING#'';
   instHMIStationDriver.instsHSSPartSelect[4].lib.raw[45,5] := WSTRING#'';
   instHMIStationDriver.instsHSSPartSelect[4].lib.raw[45,6] := WSTRING#'';
   instHMIStationDriver.instsHSSPartSelect[4].lib.raw[45,7] := WSTRING#'';
   instHMIStationDriver.instsHSSPartSelect[4].lib.raw[46,0] := WSTRING#'';
   instHMIStationDriver.instsHSSPartSelect[4].lib.raw[46,1] := WSTRING#'';
   instHMIStationDriver.instsHSSPartSelect[4].lib.raw[46,2] := WSTRING#'';
   instHMIStationDriver.instsHSSPartSelect[4].lib.raw[46,3] := WSTRING#'';
   instHMIStationDriver.instsHSSPartSelect[4].lib.raw[46,4] := WSTRING#'';
   instHMIStationDriver.instsHSSPartSelect[4].lib.raw[46,5] := WSTRING#'';
   instHMIStationDriver.instsHSSPartSelect[4].lib.raw[46,6] := WSTRING#'';
   instHMIStationDriver.instsHSSPartSelect[4].lib.raw[46,7] := WSTRING#'';
   instHMIStationDriver.instsHSSPartSelect[4].lib.raw[47,0] := WSTRING#'';
   instHMIStationDriver.instsHSSPartSelect[4].lib.raw[47,1] := WSTRING#'';
   instHMIStationDriver.instsHSSPartSelect[4].lib.raw[47,2] := WSTRING#'';
   instHMIStationDriver.instsHSSPartSelect[4].lib.raw[47,3] := WSTRING#'';
   instHMIStationDriver.instsHSSPartSelect[4].lib.raw[47,4] := WSTRING#'';
   instHMIStationDriver.instsHSSPartSelect[4].lib.raw[47,5] := WSTRING#'';
   instHMIStationDriver.instsHSSPartSelect[4].lib.raw[47,6] := WSTRING#'';
   instHMIStationDriver.instsHSSPartSelect[4].lib.raw[47,7] := WSTRING#'';
   instHMIStationDriver.instsHSSPartSelect[4].lib.raw[48,0] := WSTRING#'';
   instHMIStationDriver.instsHSSPartSelect[4].lib.raw[48,1] := WSTRING#'';
   instHMIStationDriver.instsHSSPartSelect[4].lib.raw[48,2] := WSTRING#'';
   instHMIStationDriver.instsHSSPartSelect[4].lib.raw[48,3] := WSTRING#'';
   instHMIStationDriver.instsHSSPartSelect[4].lib.raw[48,4] := WSTRING#'';
   instHMIStationDriver.instsHSSPartSelect[4].lib.raw[48,5] := WSTRING#'';
   instHMIStationDriver.instsHSSPartSelect[4].lib.raw[48,6] := WSTRING#'';
   instHMIStationDriver.instsHSSPartSelect[4].lib.raw[48,7] := WSTRING#'';
   instHMIStationDriver.instsHSSPartSelect[4].lib.raw[49,0] := WSTRING#'';
   instHMIStationDriver.instsHSSPartSelect[4].lib.raw[49,1] := WSTRING#'';
   instHMIStationDriver.instsHSSPartSelect[4].lib.raw[49,2] := WSTRING#'';
   instHMIStationDriver.instsHSSPartSelect[4].lib.raw[49,3] := WSTRING#'';
   instHMIStationDriver.instsHSSPartSelect[4].lib.raw[49,4] := WSTRING#'';
   instHMIStationDriver.instsHSSPartSelect[4].lib.raw[49,5] := WSTRING#'';
   instHMIStationDriver.instsHSSPartSelect[4].lib.raw[49,6] := WSTRING#'';
   instHMIStationDriver.instsHSSPartSelect[4].lib.raw[49,7] := WSTRING#'';
   tmrResetTimers.ST := T#-8D_9H_55M_34S_108MS;
   tmrResetTimers.PT := T#10S;
END_DATA_BLOCK

DATA_BLOCK "HMI"   // DB2
{ S7_Optimized_Access := 'TRUE' }
VERSION : 0.1
   VAR
      barcode : "Barcode Screen";
      networkHealth : "Network Health Screen";
      partCall : "Part Call Screen";
      screenNumber : Int;
      settings : "Settings";
      simStations : "Simulated Stations";
      tableNav : "Table Nav";
   END_VAR
BEGIN
END_DATA_BLOCK

DATA_BLOCK "Parts"   // DB3
{ S7_Optimized_Access := 'TRUE' }
VERSION : 0.1
   VAR RETAIN
      pRow : Int;
      requests : "Part Request Data";
   END_VAR
BEGIN
END_DATA_BLOCK

DATA_BLOCK "LED Sign"   // DB4
{ S7_Optimized_Access := 'TRUE' }
VERSION : 0.1
   VAR
      request : "LED Sign Data";
   END_VAR
BEGIN
END_DATA_BLOCK

DATA_BLOCK "Log Buffer"   // DB5
{ S7_Optimized_Access := 'TRUE' }
VERSION : 0.1
   VAR RETAIN
      logFlag : Int;
      partReq : "Part Req Log";
   END_VAR
BEGIN
END_DATA_BLOCK

DATA_BLOCK "HMI Select Stations"   // DB6
{ S7_Optimized_Access := 'TRUE' }
VERSION : 0.1
   VAR
      me : Array[0.."hmiStnCount"] of "HSS: Compressed";
   END_VAR
BEGIN
END_DATA_BLOCK

DATA_BLOCK "Net Diag: Global"   // DB7
{ S7_Optimized_Access := 'TRUE' }
VERSION : 0.1
   VAR
      plcData : "UserDiag_typePLC";   // PLC diagnostics data
      ioSystemData : Array[1.."USERDIAG_IO_SYSTEMS_UPPER_LIM"] of "UserDiag_typeIOSystem";   // IO-System diagnostics data
      startDiag : Bool := false;   // Startflag for diagnostic
   END_VAR
BEGIN
END_DATA_BLOCK

DATA_BLOCK "Net Diag: Startup"   // DB8
{ S7_Optimized_Access := 'TRUE' }
VERSION : 0.1
// stored: InstanceOfName NetDiag: Coordinate
"NetDiag: Coordinate"
BEGIN
END_DATA_BLOCK

